// TwinCAT 3 PLC project PLC
// ProgramVersion: 3.1.4023.0
// libraries:
//   Tc2_Standard, * (Beckhoff Automation GmbH)
//   Tc2_System, * (Beckhoff Automation GmbH)
//   Tc3_Module, * (Beckhoff Automation GmbH)
// project tree:
//   / PlcTask.TcTTO
//   POUs/ MAIN.TcPOU
//   DUTs/IO/PdoEntries/ Status_9847B4EF.TcDUT, Status_BA3D1C5D.TcDUT, Status_F2CE6D91.TcDUT, Control_EBEDCF76.TcDUT, FSOE_BBDEEE9E.TcDUT, FSOE_BAC7BF21.TcDUT, FSOE_39DE0EE0.TcDUT, FSOE_3E4279E1.TcDUT, FSOE_BAA7477B.TcDUT, FSOE_CEFF8C56.TcDUT, FSOE_E251F244.TcDUT, FSOE_CDFABDDF.TcDUT
//   DUTs/IO/PDOs/ InfoData_6F19DB2B.TcDUT, ID_07C9D28F.TcDUT, WcState_9091E0EB.TcDUT, Status_Us_B1E819A2.TcDUT, Status_Up_B1E819A2.TcDUT, Channel_830843C1.TcDUT, Channel_42CA91F7.TcDUT, WcState_0B2B16F9.TcDUT, MMS_Device_Inputs_ADC3123E.TcDUT, MMS_Acceleration_Status_11769099.TcDUT, MMS_Acceleration_X_Axis_80E77D6A.TcDUT, MMS_Acceleration_Y_Axis_80E77D6A.TcDUT, MMS_Acceleration_Z_Axis_80E77D6A.TcDUT, MMS_Acceleration_Timestamp_8B9FE1A2.TcDUT, MMS_Voltage_Us_In_Inputs_60D55C72.TcDUT, MMS_Voltage_Up_In_Inputs_60D55C72.TcDUT, MMS_Voltage_Up_Out_Inputs_60D55C72.TcDUT, MMS_Device_Outputs_E6E6F9D1.TcDUT, InfoData_BEF6B88E.TcDUT, FSoE_Inputs_9283FC69.TcDUT, FSoE_Outputs_79E75DAB.TcDUT, Outputs_63C46CC8.TcDUT, FSLOGIC_Inputs_EEE9388E.TcDUT, EMPTY_STRUCTURE.TcDUT, WcState_B516A264.TcDUT, InfoData_32EB74EA.TcDUT, Module_1_FSoE_BE928FF7.TcDUT, Module_2_FSOUT_E84B1B00.TcDUT, Module_3_FSLOGIC_DEAB4522.TcDUT, FSoE_Inputs_6CB74C4A.TcDUT, FSoE_Outputs_D8082339.TcDUT, Outputs_D994E0F9.TcDUT, Module_1_FSoE_042BAFD3.TcDUT, Module_2_FSOUT_8B7AA8A2.TcDUT, FSoE_Inputs_905C1934.TcDUT, FSoE_Outputs_77F9785A.TcDUT, Module_1_FSoE_7E6C60DE.TcDUT, FSoE_Inputs_A1F422BE.TcDUT, FSoE_Outputs_37DEC564.TcDUT, Module_1_FSoE_B78AD590.TcDUT, InfoData_E68C61CD.TcDUT, InfoData_2A97D6CF.TcDUT, Inputs_25A0042B.TcDUT, Outputs_2397A10E.TcDUT
//   DUTs/IO/Boxes/ EK1100_1FC0878B.TcDUT, EK1122_1FC0878B.TcDUT, EK1101_957D888F.TcDUT, EK1110_1FC0878B.TcDUT, EK1121_1FC0878B.TcDUT, EK1200_013D0B49.TcDUT, EK1300_6BC01D14.TcDUT, EK1322_6BC01D14.TcDUT, EK1310_6BC01D14.TcDUT, EK1501_957D888F.TcDUT, EK1541_957D888F.TcDUT, EK1561_1FC0878B.TcDUT, EK1521_1FC0878B.TcDUT, EK1814_F6D9A8D1.TcDUT, EK1818_6B19C24E.TcDUT, EK1828_56D6F887.TcDUT, EK1828_E2806B95.TcDUT, EKM1101_7F417622.TcDUT, EK1960_14394C51.TcDUT, EK1960_9900B192.TcDUT, EK1960_BAE25DEC.TcDUT, EK1960_2415CDAE.TcDUT
//   DUTs/IO/Devices/ SyncUnitTask_2D604ED5.TcDUT, SyncUnitTasks_6FEB8257.TcDUT, SyncUnits_99E584AF.TcDUT
//   DUTs/IO/Topology/ Beckhoff_EK11xxEK1122_42F1D1D1.TcDUT, Beckhoff_EK11xx_811529C6.TcDUT, Beckhoff_EK12xxEK1122_F8B8118B.TcDUT, Beckhoff_EK12xx_F07DE953.TcDUT, Beckhoff_EK13xxEK1122_30D1B042.TcDUT, Beckhoff_EK13xx_7663BCA8.TcDUT, Beckhoff_EK15xxEK1122_1A424B62.TcDUT, Beckhoff_EK15xx_47CB6E2F.TcDUT, Beckhoff_EK18xxEK1122_F7FACD4D.TcDUT, Beckhoff_EK18xx_88ED272B.TcDUT, Beckhoff_EKM1xxxEK1122_F03648A5.TcDUT, Beckhoff_EKM1xxx_245084ED.TcDUT, Beckhoff_EKx9xxEK1122_41BF98AA.TcDUT, Beckhoff_EKx9xx_36A98EAE.TcDUT, Beckhoff_EKxxxx_0080EK1122_9CBA35F2.TcDUT, Beckhoff_EKxxxx_0080_9DDEF925.TcDUT, EtherCAT_Master_EKxxxx_2095F716.TcDUT
//   DUTs/IO/Base/ EtcSlaveBase_82538BE2.TcDUT, EtcSlaveBase_82538BE2.TcDUT, EtcSlaveBase_82538BE2.TcDUT, EtcSlaveTerminalBase_947E5A46.TcDUT, EtcSlaveBoxBase_77A0E4A7.TcDUT, EtcSlaveEndTerminalBase_866C7F0C.TcDUT, InputBase_8311D824.TcDUT, OutputBase_10CEE7DE.TcDUT, EtcMasterBase_62654B43.TcDUT
//   GVLs/ GVL_iXlinker.TcGVL
// real-time tasks:
//   TASK PlcTask: cycle T#10ms, priority 20, ADS port 350
// I/O:
//   DEVICE EtherCAT_Master_EKxxxx, AmsNetId 172.20.30.238.8.1
//     Beckhoff EK11xx [EK1100 EtherCAT Coupler (2A E-Bus)]
//       Beckhoff EK11xxEK1122 [EK1122 2 port EtherCAT junction]
//         Beckhoff EK11xxsub EK1100 [EK1100 EtherCAT Coupler (2A E-Bus)]
//         A_0001(EK1100-0000-0000) [EK1100 EtherCAT Coupler (0.5A E-Bus)]
//         A_0002(EK1100-0000-0001) [EK1100 EtherCAT Coupler (2A E-Bus)]
//         A_0003(EK1100-0000-0016) [EK1100 EtherCAT Coupler (2A E-Bus)]
//         A_0004(EK1100-0000-0017) [EK1100 EtherCAT Coupler (2A E-Bus)]
//         A_0005(EK1100-0000-0018) [EK1100 EtherCAT Coupler (2A E-Bus)]
//         A_0006(EK1100-0008-0016) [EK1100-0008 EtherCAT Coupler M8 (2A E-Bus)]
//         A_0009(EK1101-0000-0016) [EK1101 EtherCAT Coupler (2A E-Bus, ID switch)]
//         A_0010(EK1101-0000-0017) [EK1101 EtherCAT Coupler (2A E-Bus, ID switch)]
//         A_0011(EK1101-0000-0018) [EK1101 EtherCAT Coupler (2A E-Bus, ID switch)]
//         A_0012(EK1101-0008-0016) [EK1101-0008 EtherCAT Coupler M8 (2A E-Bus, ID switch)]
//         A_0013(EK1101-0010-0016) [EK1101-0010 EtherCAT Coupler (2A E-Bus, ID switch, Extended Distance)]
//         A_0008(EK1100-0030-0017) [EK1100-0030 EtherCAT Coupler (2A E-Bus, 4kV galv. iso.)]
//         A_0007(EK1100-0030-0016) [EK1100-0030 EtherCAT Coupler (2A E-Bus, 4kV galv. iso.)]
//       A_0018(EK1110-0043-0016) [EK1110-0043 EtherCAT EJ coupler]
//       A_0024(EK1122-0008-0016) [EK1122-0008 2 port EtherCAT junction M8]
//       A_0023(EK1122-0000-0018) [EK1122 2 port EtherCAT junction]
//       A_0022(EK1122-0000-0017) [EK1122 2 port EtherCAT junction]
//       A_0021(EK1122-0000-0016) [EK1122 2 port EtherCAT junction]
//       A_0020(EK1121-0010-0016) [EK1121-0010 1 port EtherCAT junction (Extended Distance)]
//       A_0019(EK1110-0044-0016) [EK1110-0044 EtherCAT EJ coupler]
//       A_0017(EK1110-0008-0016) [EK1110-0008 EtherCAT extension M8]
//       A_0016(EK1110-0000-0017) [EK1110 EtherCAT extension]
//       A_0015(EK1110-0000-0016) [EK1110 EtherCAT extension]
//       A_0014(EK1110-0000-0000) [EK1110 EtherCAT extension]
//     Beckhoff EK12xx [EK1100 EtherCAT Coupler (2A E-Bus)]
//       Beckhoff EK12xxEK1122 [EK1122 2 port EtherCAT junction]
//         Beckhoff EK12xxsub EK1100 [EK1100 EtherCAT Coupler (2A E-Bus)]
//         A_0002(EK1200-7000-0000) [EK1200-7000 EtherCAT Power supply (1,5A E-Bus)]
//         A_0001(EK1200-5000-0000) [EK1200-5000 EtherCAT Power supply (2A E-Bus)]
//     Beckhoff EK13xx [EK1100 EtherCAT Coupler (2A E-Bus)]
//       Beckhoff EK13xxEK1122 [EK1122 2 port EtherCAT junction]
//         Beckhoff EK13xxsub EK1100 [EK1100 EtherCAT Coupler (2A E-Bus)]
//         A_0001(EK1300-0000-0017) [EK1300 EtherCAT P Coupler (2A E-Bus)]
//       A_0003(EK1322-0000-0017) [EK1322 2-port EtherCAT P junction with feed-in]
//       A_0002(EK1310-0000-0017) [EK1310 EtherCAT P extension with feed-in]
//     Beckhoff EK15xx [EK1100 EtherCAT Coupler (2A E-Bus)]
//       Beckhoff EK15xxEK1122 [EK1122 2 port EtherCAT junction]
//         Beckhoff EK15xxsub EK1100 [EK1100 EtherCAT Coupler (2A E-Bus)]
//         A_0001(EK1501-0000-0016) [EK1501 EtherCAT Coupler (2A E-Bus, FX-MultiMode, ID switch)]
//         A_0002(EK1501-0000-0017) [EK1501 EtherCAT Coupler (2A E-Bus, FX-MultiMode, ID switch)]
//         A_0003(EK1501-0000-0018) [EK1501 EtherCAT Coupler (2A E-Bus, FX-MultiMode, ID switch)]
//         A_0004(EK1501-0000-0019) [EK1501 EtherCAT Coupler (2A E-Bus, FX-MultiMode, ID switch)]
//         A_0005(EK1501-0010-0016) [EK1501-0010 EtherCAT Coupler (2A E-Bus, FX-SingleMode, ID switch)]
//         A_0006(EK1501-0010-0017) [EK1501-0010 EtherCAT Coupler (2A E-Bus, FX-SingleMode, ID switch)]
//         A_0007(EK1501-0010-0018) [EK1501-0010 EtherCAT Coupler (2A E-Bus, FX-SingleMode, ID switch)]
//         A_0008(EK1501-0100-0016) [EK1501-0100 EtherCAT Coupler (2A E-Bus, FX-MultiMode, media converter, ID switch)]
//         A_0020(EK1541-0000-0016) [EK1541 EtherCAT Coupler (2A E-Bus, POF, ID switch)]
//         A_0021(EK1541-0000-0017) [EK1541 EtherCAT Coupler (2A E-Bus, POF, ID switch)]
//         A_0022(EK1541-0000-0018) [EK1541 EtherCAT Coupler (2A E-Bus, POF, ID switch)]
//       A_0025(EK1561-0000-0018) [EK1561 1 port EtherCAT junction (POF)]
//       A_0024(EK1561-0000-0017) [EK1561 1 port EtherCAT junction (POF)]
//       A_0023(EK1561-0000-0016) [EK1561 1 port EtherCAT junction (POF)]
//       A_0019(EK1521-0010-0020) [EK1521-0010 1 port EtherCAT junction (FX-SingleMode)]
//       A_0018(EK1521-0010-0019) [EK1521-0010 1 port EtherCAT junction (FX-SingleMode)]
//       A_0017(EK1521-0010-0018) [EK1521-0010 1 port EtherCAT junction (FX-SingleMode)]
//       A_0016(EK1521-0010-0017) [EK1521-0010 1 port EtherCAT junction (FX-SingleMode)]
//       A_0015(EK1521-0010-0016) [EK1521-0010 1 port EtherCAT junction (FX-SingleMode)]
//       A_0014(EK1521-0000-0021) [EK1521 1 port EtherCAT junction (FX-MultiMode)]
//       A_0013(EK1521-0000-0020) [EK1521 1 port EtherCAT junction (FX-MultiMode)]
//       A_0012(EK1521-0000-0019) [EK1521 1 port EtherCAT junction (FX-MultiMode)]
//       A_0011(EK1521-0000-0018) [EK1521 1 port EtherCAT junction (FX-MultiMode)]
//       A_0010(EK1521-0000-0017) [EK1521 1 port EtherCAT junction (FX-MultiMode)]
//       A_0009(EK1521-0000-0016) [EK1521 1 port EtherCAT junction (FX-MultiMode)]
//     Beckhoff EK18xx [EK1100 EtherCAT Coupler (2A E-Bus)]
//       Beckhoff EK18xxEK1122 [EK1122 2 port EtherCAT junction]
//         Beckhoff EK18xxsub EK1100 [EK1100 EtherCAT Coupler (2A E-Bus)]
//         A_0001(EK1814-0000-0016) [EK1814 EtherCAT IO-Coupler  (0,5A E-Bus, 4 Ch. Dig. In, 3ms, 4 Ch. Dig. Out 24V, 0,5A)]
//         A_0002(EK1814-0000-0017) [EK1814 EtherCAT IO-Coupler  (1A E-Bus, 4 Ch. Dig. In, 3ms, 4 Ch. Dig. Out 24V, 0,5A)]
//         A_0003(EK1814-0000-0018) [EK1814 EtherCAT IO-Coupler  (1A E-Bus, 4 Ch. Dig. In, 3ms, 4 Ch. Dig. Out 24V, 0,5A)]
//         A_0004(EK1814-0000-0019) [EK1814 EtherCAT IO-Coupler  (1A E-Bus, 4 Ch. Dig. In, 3ms, 4 Ch. Dig. Out 24V, 0,5A)]
//         A_0005(EK1818-0000-0016) [EK1818 EtherCAT IO-Coupler  (1A E-Bus, 8 Ch. Dig. In, 3ms, 4 Ch. Dig. Out 24V, 0,5A)]
//         A_0006(EK1818-0000-0017) [EK1818 EtherCAT IO-Coupler  (1A E-Bus, 8 Ch. Dig. In, 3ms, 4 Ch. Dig. Out 24V, 0,5A)]
//         A_0007(EK1818-0000-0018) [EK1818 EtherCAT IO-Coupler  (1A E-Bus, 8 Ch. Dig. In, 3ms, 4 Ch. Dig. Out 24V, 0,5A)]
//         A_0008(EK1828-0000-0016) [EK1828 EtherCAT IO-Coupler  (1A E-Bus, 4 Ch. Dig. In, 3ms, 8 Ch. Dig. Out 24V, 0,5A)]
//         A_0009(EK1828-0000-0017) [EK1828 EtherCAT IO-Coupler  (1A E-Bus, 4 Ch. Dig. In, 3ms, 8 Ch. Dig. Out 24V, 0,5A)]
//         A_0010(EK1828-0000-0018) [EK1828 EtherCAT IO-Coupler  (1A E-Bus, 4 Ch. Dig. In, 3ms, 8 Ch. Dig. Out 24V, 0,5A)]
//         A_0011(EK1828-0010-0016) [EK1828-0010 EtherCAT IO-Coupler  (1A E-Bus, 8 Ch. Dig. Out 24V, 0,5A)]
//         A_0012(EK1828-0010-0017) [EK1828-0010 EtherCAT IO-Coupler  (1A E-Bus, 8 Ch. Dig. Out 24V, 0,5A)]
//         A_0013(EK1828-0010-0018) [EK1828-0010 EtherCAT IO-Coupler  (1A E-Bus, 8 Ch. Dig. Out 24V, 0,5A)]
//     Beckhoff EKM1xxx [EK1100 EtherCAT Coupler (2A E-Bus)]
//       Beckhoff EKM1xxxEK1122 [EK1122 2 port EtherCAT junction]
//         Beckhoff EKM1xxxsub EK1100 [EK1100 EtherCAT Coupler (2A E-Bus)]
//         A_0001(EKM1101-0000-0016) [EKM1101 EtherCAT Coupler  (2A E-Bus, ID switch, Diagnostics, isolated)]
//         A_0002(EKM1101-0000-0017) [EKM1101 EtherCAT Coupler  (2A E-Bus, ID switch, Diagnostics, isolated)]
//         A_0003(EKM1101-0000-0018) [EKM1101 EtherCAT Coupler  (2A E-Bus, ID switch, Diagnostics, isolated)]
//         A_0004(EKM1101-0000-0019) [EKM1101 EtherCAT Coupler  (2A E-Bus, ID switch, Diagnostics, isolated)]
//         A_0005(EKM1101-0000-0020) [EKM1101 EtherCAT Coupler  (2A E-Bus, ID switch, Diagnostics, isolated)]
//     Beckhoff EKx9xx [EK1100 EtherCAT Coupler (2A E-Bus)]
//       Beckhoff EKx9xxEK1122 [EK1122 2 port EtherCAT junction]
//         Beckhoff EKx9xxsub EK1100 [EK1100 EtherCAT Coupler (2A E-Bus)]
//         A_0001(EK1960-0000-0019) [EK1960-0000 TwinSAFE-Compact-Controller (RJ45)]
//           modules: Module 1 (FSoE), Module 2 (FSOUT), Module 3 (FSLOGIC)
//         A_0002(EK1960-0000-0021) [EK1960-0000 TwinSAFE-Compact-Controller (RJ45)]
//           modules: Module 1 (FSoE), Module 2 (FSOUT), Module 3 (FSLOGIC)
//         A_0003(EK1960-0008-0019) [EK1960-0008 TwinSAFE-Compact-Controller (M8)]
//           modules: Module 1 (FSoE), Module 2 (FSOUT), Module 3 (FSLOGIC)
//         A_0004(EK1960-0008-0021) [EK1960-0008 TwinSAFE-Compact-Controller (M8)]
//           modules: Module 1 (FSoE), Module 2 (FSOUT), Module 3 (FSLOGIC)
//         A_0005(EK1960-2600-0019) [EK1960-2600 TwinSAFE-Compact-Controller (4 x Relay, RJ45)]
//           modules: Module 1 (FSoE), Module 2 (FSOUT), Module 3 (FSLOGIC)
//         A_0006(EK1960-2600-0021) [EK1960-2600 TwinSAFE-Compact-Controller (4 x Relay, RJ45)]
//           modules: Module 1 (FSoE), Module 2 (FSOUT), Module 3 (FSLOGIC)
//         A_0007(EK1960-2608-0019) [EK1960-2608 TwinSAFE-Compact-Controller (4 x Relay, M8)]
//           modules: Module 1 (FSoE), Module 2 (FSOUT), Module 3 (FSLOGIC)
//         A_0008(EK1960-2608-0021) [EK1960-2608 TwinSAFE-Compact-Controller (4 x Relay, M8)]
//           modules: Module 1 (FSoE), Module 2 (FSOUT), Module 3 (FSLOGIC)
//     Beckhoff EKxxxx-0080 [EK1100 EtherCAT Coupler (2A E-Bus)]
//       Beckhoff EKxxxx-0080EK1122 [EK1122 2 port EtherCAT junction]
//         Beckhoff EKxxxx-0080sub EK1100 [EK1100 EtherCAT Coupler (2A E-Bus)]
//       A_0006(EK1122-0080-0019) [EK1122-0080 2 port EtherCAT junction (Fast Hot Connect)]
//       A_0005(EK1122-0080-0018) [EK1122-0080 2 port EtherCAT junction (Fast Hot Connect)]
//       A_0004(EK1122-0080-0017) [EK1122-0080 2 port EtherCAT junction (Fast Hot Connect)]
// variable links:
//   PLC/PLC Instance <-> EtherCAT Master EKxxxx/Beckhoff EK11xx
//     PlcTask Inputs/GVL_iXlinker.EtherCAT_Master_EKxxxx.Beckhoff_EK11xx.InfoData.State <-> InfoData/State
//   PLC/PLC Instance <-> EtherCAT Master EKxxxx/Beckhoff EK11xx/Beckhoff EK11xxEK1122
//     PlcTask Inputs/GVL_iXlinker.EtherCAT_Master_EKxxxx.Beckhoff_EK11xx.Beckhoff_EK11xxEK1122.InfoData.State <-> InfoData/State
//   PLC/PLC Instance <-> EtherCAT Master EKxxxx/Beckhoff EK11xx/Beckhoff EK11xxEK1122/Beckhoff EK11xxsub EK1100
//     PlcTask Inputs/GVL_iXlinker.EtherCAT_Master_EKxxxx.Beckhoff_EK11xx.Beckhoff_EK11xxEK1122.Beckhoff_EK11xxsub_EK1100.InfoData.State <-> InfoData/State
//   PLC/PLC Instance <-> EtherCAT Master EKxxxx/Beckhoff EK11xx/Beckhoff EK11xxEK1122/A_0001(EK1100-0000-0000)
//     PlcTask Inputs/GVL_iXlinker.EtherCAT_Master_EKxxxx.Beckhoff_EK11xx.Beckhoff_EK11xxEK1122.A_0001_EK1100_0000_0000.InfoData.State <-> InfoData/State
//   PLC/PLC Instance <-> EtherCAT Master EKxxxx/Beckhoff EK11xx/Beckhoff EK11xxEK1122/A_0002(EK1100-0000-0001)
//     PlcTask Inputs/GVL_iXlinker.EtherCAT_Master_EKxxxx.Beckhoff_EK11xx.Beckhoff_EK11xxEK1122.A_0002_EK1100_0000_0001.InfoData.State <-> InfoData/State
//   PLC/PLC Instance <-> EtherCAT Master EKxxxx/Beckhoff EK11xx/Beckhoff EK11xxEK1122/A_0003(EK1100-0000-0016)
//     PlcTask Inputs/GVL_iXlinker.EtherCAT_Master_EKxxxx.Beckhoff_EK11xx.Beckhoff_EK11xxEK1122.A_0003_EK1100_0000_0016.InfoData.State <-> InfoData/State
//   PLC/PLC Instance <-> EtherCAT Master EKxxxx/Beckhoff EK11xx/Beckhoff EK11xxEK1122/A_0004(EK1100-0000-0017)
//     PlcTask Inputs/GVL_iXlinker.EtherCAT_Master_EKxxxx.Beckhoff_EK11xx.Beckhoff_EK11xxEK1122.A_0004_EK1100_0000_0017.InfoData.State <-> InfoData/State
//   PLC/PLC Instance <-> EtherCAT Master EKxxxx/Beckhoff EK11xx/Beckhoff EK11xxEK1122/A_0005(EK1100-0000-0018)
//     PlcTask Inputs/GVL_iXlinker.EtherCAT_Master_EKxxxx.Beckhoff_EK11xx.Beckhoff_EK11xxEK1122.A_0005_EK1100_0000_0018.InfoData.State <-> InfoData/State
//   PLC/PLC Instance <-> EtherCAT Master EKxxxx/Beckhoff EK11xx/Beckhoff EK11xxEK1122/A_0006(EK1100-0008-0016)
//     PlcTask Inputs/GVL_iXlinker.EtherCAT_Master_EKxxxx.Beckhoff_EK11xx.Beckhoff_EK11xxEK1122.A_0006_EK1100_0008_0016.InfoData.State <-> InfoData/State
//   PLC/PLC Instance <-> EtherCAT Master EKxxxx/Beckhoff EK11xx/Beckhoff EK11xxEK1122/A_0009(EK1101-0000-0016)
//     PlcTask Inputs/GVL_iXlinker.EtherCAT_Master_EKxxxx.Beckhoff_EK11xx.Beckhoff_EK11xxEK1122.A_0009_EK1101_0000_0016.ID.ID <-> ID/ID
//     PlcTask Inputs/GVL_iXlinker.EtherCAT_Master_EKxxxx.Beckhoff_EK11xx.Beckhoff_EK11xxEK1122.A_0009_EK1101_0000_0016.WcState.WcState <-> WcState/WcState
//     PlcTask Inputs/GVL_iXlinker.EtherCAT_Master_EKxxxx.Beckhoff_EK11xx.Beckhoff_EK11xxEK1122.A_0009_EK1101_0000_0016.WcState.InputToggle <-> WcState/InputToggle
//     PlcTask Inputs/GVL_iXlinker.EtherCAT_Master_EKxxxx.Beckhoff_EK11xx.Beckhoff_EK11xxEK1122.A_0009_EK1101_0000_0016.InfoData.State <-> InfoData/State
//   PLC/PLC Instance <-> EtherCAT Master EKxxxx/Beckhoff EK11xx/Beckhoff EK11xxEK1122/A_0010(EK1101-0000-0017)
//     PlcTask Inputs/GVL_iXlinker.EtherCAT_Master_EKxxxx.Beckhoff_EK11xx.Beckhoff_EK11xxEK1122.A_0010_EK1101_0000_0017.ID.ID <-> ID/ID
//     PlcTask Inputs/GVL_iXlinker.EtherCAT_Master_EKxxxx.Beckhoff_EK11xx.Beckhoff_EK11xxEK1122.A_0010_EK1101_0000_0017.WcState.WcState <-> WcState/WcState
//     PlcTask Inputs/GVL_iXlinker.EtherCAT_Master_EKxxxx.Beckhoff_EK11xx.Beckhoff_EK11xxEK1122.A_0010_EK1101_0000_0017.WcState.InputToggle <-> WcState/InputToggle
//     PlcTask Inputs/GVL_iXlinker.EtherCAT_Master_EKxxxx.Beckhoff_EK11xx.Beckhoff_EK11xxEK1122.A_0010_EK1101_0000_0017.InfoData.State <-> InfoData/State
//   PLC/PLC Instance <-> EtherCAT Master EKxxxx/Beckhoff EK11xx/Beckhoff EK11xxEK1122/A_0011(EK1101-0000-0018)
//     PlcTask Inputs/GVL_iXlinker.EtherCAT_Master_EKxxxx.Beckhoff_EK11xx.Beckhoff_EK11xxEK1122.A_0011_EK1101_0000_0018.ID.ID <-> ID/ID
//     PlcTask Inputs/GVL_iXlinker.EtherCAT_Master_EKxxxx.Beckhoff_EK11xx.Beckhoff_EK11xxEK1122.A_0011_EK1101_0000_0018.WcState.WcState <-> WcState/WcState
//     PlcTask Inputs/GVL_iXlinker.EtherCAT_Master_EKxxxx.Beckhoff_EK11xx.Beckhoff_EK11xxEK1122.A_0011_EK1101_0000_0018.WcState.InputToggle <-> WcState/InputToggle
//     PlcTask Inputs/GVL_iXlinker.EtherCAT_Master_EKxxxx.Beckhoff_EK11xx.Beckhoff_EK11xxEK1122.A_0011_EK1101_0000_0018.InfoData.State <-> InfoData/State
//   PLC/PLC Instance <-> EtherCAT Master EKxxxx/Beckhoff EK11xx/Beckhoff EK11xxEK1122/A_0012(EK1101-0008-0016)
//     PlcTask Inputs/GVL_iXlinker.EtherCAT_Master_EKxxxx.Beckhoff_EK11xx.Beckhoff_EK11xxEK1122.A_0012_EK1101_0008_0016.ID.ID <-> ID/ID
//     PlcTask Inputs/GVL_iXlinker.EtherCAT_Master_EKxxxx.Beckhoff_EK11xx.Beckhoff_EK11xxEK1122.A_0012_EK1101_0008_0016.WcState.WcState <-> WcState/WcState
//     PlcTask Inputs/GVL_iXlinker.EtherCAT_Master_EKxxxx.Beckhoff_EK11xx.Beckhoff_EK11xxEK1122.A_0012_EK1101_0008_0016.WcState.InputToggle <-> WcState/InputToggle
//     PlcTask Inputs/GVL_iXlinker.EtherCAT_Master_EKxxxx.Beckhoff_EK11xx.Beckhoff_EK11xxEK1122.A_0012_EK1101_0008_0016.InfoData.State <-> InfoData/State
//   PLC/PLC Instance <-> EtherCAT Master EKxxxx/Beckhoff EK11xx/Beckhoff EK11xxEK1122/A_0013(EK1101-0010-0016)
//     PlcTask Inputs/GVL_iXlinker.EtherCAT_Master_EKxxxx.Beckhoff_EK11xx.Beckhoff_EK11xxEK1122.A_0013_EK1101_0010_0016.ID.ID <-> ID/ID
//     PlcTask Inputs/GVL_iXlinker.EtherCAT_Master_EKxxxx.Beckhoff_EK11xx.Beckhoff_EK11xxEK1122.A_0013_EK1101_0010_0016.WcState.WcState <-> WcState/WcState
//     PlcTask Inputs/GVL_iXlinker.EtherCAT_Master_EKxxxx.Beckhoff_EK11xx.Beckhoff_EK11xxEK1122.A_0013_EK1101_0010_0016.WcState.InputToggle <-> WcState/InputToggle
//     PlcTask Inputs/GVL_iXlinker.EtherCAT_Master_EKxxxx.Beckhoff_EK11xx.Beckhoff_EK11xxEK1122.A_0013_EK1101_0010_0016.InfoData.State <-> InfoData/State
//   PLC/PLC Instance <-> EtherCAT Master EKxxxx/Beckhoff EK11xx/Beckhoff EK11xxEK1122/A_0008(EK1100-0030-0017)
//     PlcTask Inputs/GVL_iXlinker.EtherCAT_Master_EKxxxx.Beckhoff_EK11xx.Beckhoff_EK11xxEK1122.A_0008_EK1100_0030_0017.InfoData.State <-> InfoData/State
//   PLC/PLC Instance <-> EtherCAT Master EKxxxx/Beckhoff EK11xx/Beckhoff EK11xxEK1122/A_0007(EK1100-0030-0016)
//     PlcTask Inputs/GVL_iXlinker.EtherCAT_Master_EKxxxx.Beckhoff_EK11xx.Beckhoff_EK11xxEK1122.A_0007_EK1100_0030_0016.InfoData.State <-> InfoData/State
//   PLC/PLC Instance <-> EtherCAT Master EKxxxx/Beckhoff EK11xx/A_0018(EK1110-0043-0016)
//     PlcTask Inputs/GVL_iXlinker.EtherCAT_Master_EKxxxx.Beckhoff_EK11xx.A_0018_EK1110_0043_0016.InfoData.State <-> InfoData/State
//   PLC/PLC Instance <-> EtherCAT Master EKxxxx/Beckhoff EK11xx/A_0024(EK1122-0008-0016)
//     PlcTask Inputs/GVL_iXlinker.EtherCAT_Master_EKxxxx.Beckhoff_EK11xx.A_0024_EK1122_0008_0016.InfoData.State <-> InfoData/State
//   PLC/PLC Instance <-> EtherCAT Master EKxxxx/Beckhoff EK11xx/A_0023(EK1122-0000-0018)
//     PlcTask Inputs/GVL_iXlinker.EtherCAT_Master_EKxxxx.Beckhoff_EK11xx.A_0023_EK1122_0000_0018.InfoData.State <-> InfoData/State
//   PLC/PLC Instance <-> EtherCAT Master EKxxxx/Beckhoff EK11xx/A_0022(EK1122-0000-0017)
//     PlcTask Inputs/GVL_iXlinker.EtherCAT_Master_EKxxxx.Beckhoff_EK11xx.A_0022_EK1122_0000_0017.InfoData.State <-> InfoData/State
//   PLC/PLC Instance <-> EtherCAT Master EKxxxx/Beckhoff EK11xx/A_0021(EK1122-0000-0016)
//     PlcTask Inputs/GVL_iXlinker.EtherCAT_Master_EKxxxx.Beckhoff_EK11xx.A_0021_EK1122_0000_0016.InfoData.State <-> InfoData/State
//   PLC/PLC Instance <-> EtherCAT Master EKxxxx/Beckhoff EK11xx/A_0020(EK1121-0010-0016)
//     PlcTask Inputs/GVL_iXlinker.EtherCAT_Master_EKxxxx.Beckhoff_EK11xx.A_0020_EK1121_0010_0016.InfoData.State <-> InfoData/State
//   PLC/PLC Instance <-> EtherCAT Master EKxxxx/Beckhoff EK11xx/A_0019(EK1110-0044-0016)
//     PlcTask Inputs/GVL_iXlinker.EtherCAT_Master_EKxxxx.Beckhoff_EK11xx.A_0019_EK1110_0044_0016.InfoData.State <-> InfoData/State
//   PLC/PLC Instance <-> EtherCAT Master EKxxxx/Beckhoff EK11xx/A_0017(EK1110-0008-0016)
//     PlcTask Inputs/GVL_iXlinker.EtherCAT_Master_EKxxxx.Beckhoff_EK11xx.A_0017_EK1110_0008_0016.InfoData.State <-> InfoData/State
//   PLC/PLC Instance <-> EtherCAT Master EKxxxx/Beckhoff EK11xx/A_0016(EK1110-0000-0017)
//     PlcTask Inputs/GVL_iXlinker.EtherCAT_Master_EKxxxx.Beckhoff_EK11xx.A_0016_EK1110_0000_0017.InfoData.State <-> InfoData/State
//   PLC/PLC Instance <-> EtherCAT Master EKxxxx/Beckhoff EK11xx/A_0015(EK1110-0000-0016)
//     PlcTask Inputs/GVL_iXlinker.EtherCAT_Master_EKxxxx.Beckhoff_EK11xx.A_0015_EK1110_0000_0016.InfoData.State <-> InfoData/State
//   PLC/PLC Instance <-> EtherCAT Master EKxxxx/Beckhoff EK11xx/A_0014(EK1110-0000-0000)
//     PlcTask Inputs/GVL_iXlinker.EtherCAT_Master_EKxxxx.Beckhoff_EK11xx.A_0014_EK1110_0000_0000.InfoData.State <-> InfoData/State
//   PLC/PLC Instance <-> EtherCAT Master EKxxxx/Beckhoff EK12xx
//     PlcTask Inputs/GVL_iXlinker.EtherCAT_Master_EKxxxx.Beckhoff_EK12xx.InfoData.State <-> InfoData/State
//   PLC/PLC Instance <-> EtherCAT Master EKxxxx/Beckhoff EK12xx/Beckhoff EK12xxEK1122
//     PlcTask Inputs/GVL_iXlinker.EtherCAT_Master_EKxxxx.Beckhoff_EK12xx.Beckhoff_EK12xxEK1122.InfoData.State <-> InfoData/State
//   PLC/PLC Instance <-> EtherCAT Master EKxxxx/Beckhoff EK12xx/Beckhoff EK12xxEK1122/Beckhoff EK12xxsub EK1100
//     PlcTask Inputs/GVL_iXlinker.EtherCAT_Master_EKxxxx.Beckhoff_EK12xx.Beckhoff_EK12xxEK1122.Beckhoff_EK12xxsub_EK1100.InfoData.State <-> InfoData/State
//   PLC/PLC Instance <-> EtherCAT Master EKxxxx/Beckhoff EK13xx
//     PlcTask Inputs/GVL_iXlinker.EtherCAT_Master_EKxxxx.Beckhoff_EK13xx.InfoData.State <-> InfoData/State
//   PLC/PLC Instance <-> EtherCAT Master EKxxxx/Beckhoff EK13xx/Beckhoff EK13xxEK1122
//     PlcTask Inputs/GVL_iXlinker.EtherCAT_Master_EKxxxx.Beckhoff_EK13xx.Beckhoff_EK13xxEK1122.InfoData.State <-> InfoData/State
//   PLC/PLC Instance <-> EtherCAT Master EKxxxx/Beckhoff EK13xx/Beckhoff EK13xxEK1122/Beckhoff EK13xxsub EK1100
//     PlcTask Inputs/GVL_iXlinker.EtherCAT_Master_EKxxxx.Beckhoff_EK13xx.Beckhoff_EK13xxEK1122.Beckhoff_EK13xxsub_EK1100.InfoData.State <-> InfoData/State
//   PLC/PLC Instance <-> EtherCAT Master EKxxxx/Beckhoff EK13xx/Beckhoff EK13xxEK1122/A_0001(EK1300-0000-0017)
//     PlcTask Inputs/GVL_iXlinker.EtherCAT_Master_EKxxxx.Beckhoff_EK13xx.Beckhoff_EK13xxEK1122.A_0001_EK1300_0000_0017.Status_Us.Undervoltage <-> Status Us/Undervoltage
//     PlcTask Inputs/GVL_iXlinker.EtherCAT_Master_EKxxxx.Beckhoff_EK13xx.Beckhoff_EK13xxEK1122.A_0001_EK1300_0000_0017.Status_Up.Undervoltage <-> Status Up/Undervoltage
//     PlcTask Inputs/GVL_iXlinker.EtherCAT_Master_EKxxxx.Beckhoff_EK13xx.Beckhoff_EK13xxEK1122.A_0001_EK1300_0000_0017.WcState.WcState <-> WcState/WcState
//     PlcTask Inputs/GVL_iXlinker.EtherCAT_Master_EKxxxx.Beckhoff_EK13xx.Beckhoff_EK13xxEK1122.A_0001_EK1300_0000_0017.WcState.InputToggle <-> WcState/InputToggle
//     PlcTask Inputs/GVL_iXlinker.EtherCAT_Master_EKxxxx.Beckhoff_EK13xx.Beckhoff_EK13xxEK1122.A_0001_EK1300_0000_0017.InfoData.State <-> InfoData/State
//   PLC/PLC Instance <-> EtherCAT Master EKxxxx/Beckhoff EK13xx/A_0003(EK1322-0000-0017)
//     PlcTask Inputs/GVL_iXlinker.EtherCAT_Master_EKxxxx.Beckhoff_EK13xx.A_0003_EK1322_0000_0017.Status_Us.Undervoltage <-> Status Us/Undervoltage
//     PlcTask Inputs/GVL_iXlinker.EtherCAT_Master_EKxxxx.Beckhoff_EK13xx.A_0003_EK1322_0000_0017.Status_Up.Undervoltage <-> Status Up/Undervoltage
//     PlcTask Inputs/GVL_iXlinker.EtherCAT_Master_EKxxxx.Beckhoff_EK13xx.A_0003_EK1322_0000_0017.WcState.WcState <-> WcState/WcState
//     PlcTask Inputs/GVL_iXlinker.EtherCAT_Master_EKxxxx.Beckhoff_EK13xx.A_0003_EK1322_0000_0017.WcState.InputToggle <-> WcState/InputToggle
//     PlcTask Inputs/GVL_iXlinker.EtherCAT_Master_EKxxxx.Beckhoff_EK13xx.A_0003_EK1322_0000_0017.InfoData.State <-> InfoData/State
//   PLC/PLC Instance <-> EtherCAT Master EKxxxx/Beckhoff EK13xx/A_0002(EK1310-0000-0017)
//     PlcTask Inputs/GVL_iXlinker.EtherCAT_Master_EKxxxx.Beckhoff_EK13xx.A_0002_EK1310_0000_0017.Status_Us.Undervoltage <-> Status Us/Undervoltage
//     PlcTask Inputs/GVL_iXlinker.EtherCAT_Master_EKxxxx.Beckhoff_EK13xx.A_0002_EK1310_0000_0017.Status_Up.Undervoltage <-> Status Up/Undervoltage
//     PlcTask Inputs/GVL_iXlinker.EtherCAT_Master_EKxxxx.Beckhoff_EK13xx.A_0002_EK1310_0000_0017.WcState.WcState <-> WcState/WcState
//     PlcTask Inputs/GVL_iXlinker.EtherCAT_Master_EKxxxx.Beckhoff_EK13xx.A_0002_EK1310_0000_0017.WcState.InputToggle <-> WcState/InputToggle
//     PlcTask Inputs/GVL_iXlinker.EtherCAT_Master_EKxxxx.Beckhoff_EK13xx.A_0002_EK1310_0000_0017.InfoData.State <-> InfoData/State
//   PLC/PLC Instance <-> EtherCAT Master EKxxxx/Beckhoff EK15xx
//     PlcTask Inputs/GVL_iXlinker.EtherCAT_Master_EKxxxx.Beckhoff_EK15xx.InfoData.State <-> InfoData/State
//   PLC/PLC Instance <-> EtherCAT Master EKxxxx/Beckhoff EK15xx/Beckhoff EK15xxEK1122
//     PlcTask Inputs/GVL_iXlinker.EtherCAT_Master_EKxxxx.Beckhoff_EK15xx.Beckhoff_EK15xxEK1122.InfoData.State <-> InfoData/State
//   PLC/PLC Instance <-> EtherCAT Master EKxxxx/Beckhoff EK15xx/Beckhoff EK15xxEK1122/Beckhoff EK15xxsub EK1100
//     PlcTask Inputs/GVL_iXlinker.EtherCAT_Master_EKxxxx.Beckhoff_EK15xx.Beckhoff_EK15xxEK1122.Beckhoff_EK15xxsub_EK1100.InfoData.State <-> InfoData/State
//   PLC/PLC Instance <-> EtherCAT Master EKxxxx/Beckhoff EK15xx/Beckhoff EK15xxEK1122/A_0001(EK1501-0000-0016)
//     PlcTask Inputs/GVL_iXlinker.EtherCAT_Master_EKxxxx.Beckhoff_EK15xx.Beckhoff_EK15xxEK1122.A_0001_EK1501_0000_0016.ID.ID <-> ID/ID
//     PlcTask Inputs/GVL_iXlinker.EtherCAT_Master_EKxxxx.Beckhoff_EK15xx.Beckhoff_EK15xxEK1122.A_0001_EK1501_0000_0016.WcState.WcState <-> WcState/WcState
//     PlcTask Inputs/GVL_iXlinker.EtherCAT_Master_EKxxxx.Beckhoff_EK15xx.Beckhoff_EK15xxEK1122.A_0001_EK1501_0000_0016.WcState.InputToggle <-> WcState/InputToggle
//     PlcTask Inputs/GVL_iXlinker.EtherCAT_Master_EKxxxx.Beckhoff_EK15xx.Beckhoff_EK15xxEK1122.A_0001_EK1501_0000_0016.InfoData.State <-> InfoData/State
//   PLC/PLC Instance <-> EtherCAT Master EKxxxx/Beckhoff EK15xx/Beckhoff EK15xxEK1122/A_0002(EK1501-0000-0017)
//     PlcTask Inputs/GVL_iXlinker.EtherCAT_Master_EKxxxx.Beckhoff_EK15xx.Beckhoff_EK15xxEK1122.A_0002_EK1501_0000_0017.ID.ID <-> ID/ID
//     PlcTask Inputs/GVL_iXlinker.EtherCAT_Master_EKxxxx.Beckhoff_EK15xx.Beckhoff_EK15xxEK1122.A_0002_EK1501_0000_0017.WcState.WcState <-> WcState/WcState
//     PlcTask Inputs/GVL_iXlinker.EtherCAT_Master_EKxxxx.Beckhoff_EK15xx.Beckhoff_EK15xxEK1122.A_0002_EK1501_0000_0017.WcState.InputToggle <-> WcState/InputToggle
//     PlcTask Inputs/GVL_iXlinker.EtherCAT_Master_EKxxxx.Beckhoff_EK15xx.Beckhoff_EK15xxEK1122.A_0002_EK1501_0000_0017.InfoData.State <-> InfoData/State
//   PLC/PLC Instance <-> EtherCAT Master EKxxxx/Beckhoff EK15xx/Beckhoff EK15xxEK1122/A_0003(EK1501-0000-0018)
//     PlcTask Inputs/GVL_iXlinker.EtherCAT_Master_EKxxxx.Beckhoff_EK15xx.Beckhoff_EK15xxEK1122.A_0003_EK1501_0000_0018.ID.ID <-> ID/ID
//     PlcTask Inputs/GVL_iXlinker.EtherCAT_Master_EKxxxx.Beckhoff_EK15xx.Beckhoff_EK15xxEK1122.A_0003_EK1501_0000_0018.WcState.WcState <-> WcState/WcState
//     PlcTask Inputs/GVL_iXlinker.EtherCAT_Master_EKxxxx.Beckhoff_EK15xx.Beckhoff_EK15xxEK1122.A_0003_EK1501_0000_0018.WcState.InputToggle <-> WcState/InputToggle
//     PlcTask Inputs/GVL_iXlinker.EtherCAT_Master_EKxxxx.Beckhoff_EK15xx.Beckhoff_EK15xxEK1122.A_0003_EK1501_0000_0018.InfoData.State <-> InfoData/State
//   PLC/PLC Instance <-> EtherCAT Master EKxxxx/Beckhoff EK15xx/Beckhoff EK15xxEK1122/A_0004(EK1501-0000-0019)
//     PlcTask Inputs/GVL_iXlinker.EtherCAT_Master_EKxxxx.Beckhoff_EK15xx.Beckhoff_EK15xxEK1122.A_0004_EK1501_0000_0019.ID.ID <-> ID/ID
//     PlcTask Inputs/GVL_iXlinker.EtherCAT_Master_EKxxxx.Beckhoff_EK15xx.Beckhoff_EK15xxEK1122.A_0004_EK1501_0000_0019.WcState.WcState <-> WcState/WcState
//     PlcTask Inputs/GVL_iXlinker.EtherCAT_Master_EKxxxx.Beckhoff_EK15xx.Beckhoff_EK15xxEK1122.A_0004_EK1501_0000_0019.WcState.InputToggle <-> WcState/InputToggle
//     PlcTask Inputs/GVL_iXlinker.EtherCAT_Master_EKxxxx.Beckhoff_EK15xx.Beckhoff_EK15xxEK1122.A_0004_EK1501_0000_0019.InfoData.State <-> InfoData/State
//   PLC/PLC Instance <-> EtherCAT Master EKxxxx/Beckhoff EK15xx/Beckhoff EK15xxEK1122/A_0005(EK1501-0010-0016)
//     PlcTask Inputs/GVL_iXlinker.EtherCAT_Master_EKxxxx.Beckhoff_EK15xx.Beckhoff_EK15xxEK1122.A_0005_EK1501_0010_0016.ID.ID <-> ID/ID
//     PlcTask Inputs/GVL_iXlinker.EtherCAT_Master_EKxxxx.Beckhoff_EK15xx.Beckhoff_EK15xxEK1122.A_0005_EK1501_0010_0016.WcState.WcState <-> WcState/WcState
//     PlcTask Inputs/GVL_iXlinker.EtherCAT_Master_EKxxxx.Beckhoff_EK15xx.Beckhoff_EK15xxEK1122.A_0005_EK1501_0010_0016.WcState.InputToggle <-> WcState/InputToggle
//     PlcTask Inputs/GVL_iXlinker.EtherCAT_Master_EKxxxx.Beckhoff_EK15xx.Beckhoff_EK15xxEK1122.A_0005_EK1501_0010_0016.InfoData.State <-> InfoData/State
//   PLC/PLC Instance <-> EtherCAT Master EKxxxx/Beckhoff EK15xx/Beckhoff EK15xxEK1122/A_0006(EK1501-0010-0017)
//     PlcTask Inputs/GVL_iXlinker.EtherCAT_Master_EKxxxx.Beckhoff_EK15xx.Beckhoff_EK15xxEK1122.A_0006_EK1501_0010_0017.ID.ID <-> ID/ID
//     PlcTask Inputs/GVL_iXlinker.EtherCAT_Master_EKxxxx.Beckhoff_EK15xx.Beckhoff_EK15xxEK1122.A_0006_EK1501_0010_0017.WcState.WcState <-> WcState/WcState
//     PlcTask Inputs/GVL_iXlinker.EtherCAT_Master_EKxxxx.Beckhoff_EK15xx.Beckhoff_EK15xxEK1122.A_0006_EK1501_0010_0017.WcState.InputToggle <-> WcState/InputToggle
//     PlcTask Inputs/GVL_iXlinker.EtherCAT_Master_EKxxxx.Beckhoff_EK15xx.Beckhoff_EK15xxEK1122.A_0006_EK1501_0010_0017.InfoData.State <-> InfoData/State
//   PLC/PLC Instance <-> EtherCAT Master EKxxxx/Beckhoff EK15xx/Beckhoff EK15xxEK1122/A_0007(EK1501-0010-0018)
//     PlcTask Inputs/GVL_iXlinker.EtherCAT_Master_EKxxxx.Beckhoff_EK15xx.Beckhoff_EK15xxEK1122.A_0007_EK1501_0010_0018.ID.ID <-> ID/ID
//     PlcTask Inputs/GVL_iXlinker.EtherCAT_Master_EKxxxx.Beckhoff_EK15xx.Beckhoff_EK15xxEK1122.A_0007_EK1501_0010_0018.WcState.WcState <-> WcState/WcState
//     PlcTask Inputs/GVL_iXlinker.EtherCAT_Master_EKxxxx.Beckhoff_EK15xx.Beckhoff_EK15xxEK1122.A_0007_EK1501_0010_0018.WcState.InputToggle <-> WcState/InputToggle
//     PlcTask Inputs/GVL_iXlinker.EtherCAT_Master_EKxxxx.Beckhoff_EK15xx.Beckhoff_EK15xxEK1122.A_0007_EK1501_0010_0018.InfoData.State <-> InfoData/State
//   PLC/PLC Instance <-> EtherCAT Master EKxxxx/Beckhoff EK15xx/Beckhoff EK15xxEK1122/A_0008(EK1501-0100-0016)
//     PlcTask Inputs/GVL_iXlinker.EtherCAT_Master_EKxxxx.Beckhoff_EK15xx.Beckhoff_EK15xxEK1122.A_0008_EK1501_0100_0016.ID.ID <-> ID/ID
//     PlcTask Inputs/GVL_iXlinker.EtherCAT_Master_EKxxxx.Beckhoff_EK15xx.Beckhoff_EK15xxEK1122.A_0008_EK1501_0100_0016.WcState.WcState <-> WcState/WcState
//     PlcTask Inputs/GVL_iXlinker.EtherCAT_Master_EKxxxx.Beckhoff_EK15xx.Beckhoff_EK15xxEK1122.A_0008_EK1501_0100_0016.WcState.InputToggle <-> WcState/InputToggle
//     PlcTask Inputs/GVL_iXlinker.EtherCAT_Master_EKxxxx.Beckhoff_EK15xx.Beckhoff_EK15xxEK1122.A_0008_EK1501_0100_0016.InfoData.State <-> InfoData/State
//   PLC/PLC Instance <-> EtherCAT Master EKxxxx/Beckhoff EK15xx/Beckhoff EK15xxEK1122/A_0020(EK1541-0000-0016)
//     PlcTask Inputs/GVL_iXlinker.EtherCAT_Master_EKxxxx.Beckhoff_EK15xx.Beckhoff_EK15xxEK1122.A_0020_EK1541_0000_0016.ID.ID <-> ID/ID
//     PlcTask Inputs/GVL_iXlinker.EtherCAT_Master_EKxxxx.Beckhoff_EK15xx.Beckhoff_EK15xxEK1122.A_0020_EK1541_0000_0016.WcState.WcState <-> WcState/WcState
//     PlcTask Inputs/GVL_iXlinker.EtherCAT_Master_EKxxxx.Beckhoff_EK15xx.Beckhoff_EK15xxEK1122.A_0020_EK1541_0000_0016.WcState.InputToggle <-> WcState/InputToggle
//     PlcTask Inputs/GVL_iXlinker.EtherCAT_Master_EKxxxx.Beckhoff_EK15xx.Beckhoff_EK15xxEK1122.A_0020_EK1541_0000_0016.InfoData.State <-> InfoData/State
//   PLC/PLC Instance <-> EtherCAT Master EKxxxx/Beckhoff EK15xx/Beckhoff EK15xxEK1122/A_0021(EK1541-0000-0017)
//     PlcTask Inputs/GVL_iXlinker.EtherCAT_Master_EKxxxx.Beckhoff_EK15xx.Beckhoff_EK15xxEK1122.A_0021_EK1541_0000_0017.ID.ID <-> ID/ID
//     PlcTask Inputs/GVL_iXlinker.EtherCAT_Master_EKxxxx.Beckhoff_EK15xx.Beckhoff_EK15xxEK1122.A_0021_EK1541_0000_0017.WcState.WcState <-> WcState/WcState
//     PlcTask Inputs/GVL_iXlinker.EtherCAT_Master_EKxxxx.Beckhoff_EK15xx.Beckhoff_EK15xxEK1122.A_0021_EK1541_0000_0017.WcState.InputToggle <-> WcState/InputToggle
//     PlcTask Inputs/GVL_iXlinker.EtherCAT_Master_EKxxxx.Beckhoff_EK15xx.Beckhoff_EK15xxEK1122.A_0021_EK1541_0000_0017.InfoData.State <-> InfoData/State
//   PLC/PLC Instance <-> EtherCAT Master EKxxxx/Beckhoff EK15xx/Beckhoff EK15xxEK1122/A_0022(EK1541-0000-0018)
//     PlcTask Inputs/GVL_iXlinker.EtherCAT_Master_EKxxxx.Beckhoff_EK15xx.Beckhoff_EK15xxEK1122.A_0022_EK1541_0000_0018.ID.ID <-> ID/ID
//     PlcTask Inputs/GVL_iXlinker.EtherCAT_Master_EKxxxx.Beckhoff_EK15xx.Beckhoff_EK15xxEK1122.A_0022_EK1541_0000_0018.WcState.WcState <-> WcState/WcState
//     PlcTask Inputs/GVL_iXlinker.EtherCAT_Master_EKxxxx.Beckhoff_EK15xx.Beckhoff_EK15xxEK1122.A_0022_EK1541_0000_0018.WcState.InputToggle <-> WcState/InputToggle
//     PlcTask Inputs/GVL_iXlinker.EtherCAT_Master_EKxxxx.Beckhoff_EK15xx.Beckhoff_EK15xxEK1122.A_0022_EK1541_0000_0018.InfoData.State <-> InfoData/State
//   PLC/PLC Instance <-> EtherCAT Master EKxxxx/Beckhoff EK15xx/A_0025(EK1561-0000-0018)
//     PlcTask Inputs/GVL_iXlinker.EtherCAT_Master_EKxxxx.Beckhoff_EK15xx.A_0025_EK1561_0000_0018.InfoData.State <-> InfoData/State
//   PLC/PLC Instance <-> EtherCAT Master EKxxxx/Beckhoff EK15xx/A_0024(EK1561-0000-0017)
//     PlcTask Inputs/GVL_iXlinker.EtherCAT_Master_EKxxxx.Beckhoff_EK15xx.A_0024_EK1561_0000_0017.InfoData.State <-> InfoData/State
//   PLC/PLC Instance <-> EtherCAT Master EKxxxx/Beckhoff EK15xx/A_0023(EK1561-0000-0016)
//     PlcTask Inputs/GVL_iXlinker.EtherCAT_Master_EKxxxx.Beckhoff_EK15xx.A_0023_EK1561_0000_0016.InfoData.State <-> InfoData/State
//   PLC/PLC Instance <-> EtherCAT Master EKxxxx/Beckhoff EK15xx/A_0019(EK1521-0010-0020)
//     PlcTask Inputs/GVL_iXlinker.EtherCAT_Master_EKxxxx.Beckhoff_EK15xx.A_0019_EK1521_0010_0020.InfoData.State <-> InfoData/State
//   PLC/PLC Instance <-> EtherCAT Master EKxxxx/Beckhoff EK15xx/A_0018(EK1521-0010-0019)
//     PlcTask Inputs/GVL_iXlinker.EtherCAT_Master_EKxxxx.Beckhoff_EK15xx.A_0018_EK1521_0010_0019.InfoData.State <-> InfoData/State
//   PLC/PLC Instance <-> EtherCAT Master EKxxxx/Beckhoff EK15xx/A_0017(EK1521-0010-0018)
//     PlcTask Inputs/GVL_iXlinker.EtherCAT_Master_EKxxxx.Beckhoff_EK15xx.A_0017_EK1521_0010_0018.InfoData.State <-> InfoData/State
//   PLC/PLC Instance <-> EtherCAT Master EKxxxx/Beckhoff EK15xx/A_0016(EK1521-0010-0017)
//     PlcTask Inputs/GVL_iXlinker.EtherCAT_Master_EKxxxx.Beckhoff_EK15xx.A_0016_EK1521_0010_0017.InfoData.State <-> InfoData/State
//   PLC/PLC Instance <-> EtherCAT Master EKxxxx/Beckhoff EK15xx/A_0015(EK1521-0010-0016)
//     PlcTask Inputs/GVL_iXlinker.EtherCAT_Master_EKxxxx.Beckhoff_EK15xx.A_0015_EK1521_0010_0016.InfoData.State <-> InfoData/State
//   PLC/PLC Instance <-> EtherCAT Master EKxxxx/Beckhoff EK15xx/A_0014(EK1521-0000-0021)
//     PlcTask Inputs/GVL_iXlinker.EtherCAT_Master_EKxxxx.Beckhoff_EK15xx.A_0014_EK1521_0000_0021.InfoData.State <-> InfoData/State
//   PLC/PLC Instance <-> EtherCAT Master EKxxxx/Beckhoff EK15xx/A_0013(EK1521-0000-0020)
//     PlcTask Inputs/GVL_iXlinker.EtherCAT_Master_EKxxxx.Beckhoff_EK15xx.A_0013_EK1521_0000_0020.InfoData.State <-> InfoData/State
//   PLC/PLC Instance <-> EtherCAT Master EKxxxx/Beckhoff EK15xx/A_0012(EK1521-0000-0019)
//     PlcTask Inputs/GVL_iXlinker.EtherCAT_Master_EKxxxx.Beckhoff_EK15xx.A_0012_EK1521_0000_0019.InfoData.State <-> InfoData/State
//   PLC/PLC Instance <-> EtherCAT Master EKxxxx/Beckhoff EK15xx/A_0011(EK1521-0000-0018)
//     PlcTask Inputs/GVL_iXlinker.EtherCAT_Master_EKxxxx.Beckhoff_EK15xx.A_0011_EK1521_0000_0018.InfoData.State <-> InfoData/State
//   PLC/PLC Instance <-> EtherCAT Master EKxxxx/Beckhoff EK15xx/A_0010(EK1521-0000-0017)
//     PlcTask Inputs/GVL_iXlinker.EtherCAT_Master_EKxxxx.Beckhoff_EK15xx.A_0010_EK1521_0000_0017.InfoData.State <-> InfoData/State
//   PLC/PLC Instance <-> EtherCAT Master EKxxxx/Beckhoff EK15xx/A_0009(EK1521-0000-0016)
//     PlcTask Inputs/GVL_iXlinker.EtherCAT_Master_EKxxxx.Beckhoff_EK15xx.A_0009_EK1521_0000_0016.InfoData.State <-> InfoData/State
//   PLC/PLC Instance <-> EtherCAT Master EKxxxx/Beckhoff EK18xx
//     PlcTask Inputs/GVL_iXlinker.EtherCAT_Master_EKxxxx.Beckhoff_EK18xx.InfoData.State <-> InfoData/State
//   PLC/PLC Instance <-> EtherCAT Master EKxxxx/Beckhoff EK18xx/Beckhoff EK18xxEK1122
//     PlcTask Inputs/GVL_iXlinker.EtherCAT_Master_EKxxxx.Beckhoff_EK18xx.Beckhoff_EK18xxEK1122.InfoData.State <-> InfoData/State
//   PLC/PLC Instance <-> EtherCAT Master EKxxxx/Beckhoff EK18xx/Beckhoff EK18xxEK1122/Beckhoff EK18xxsub EK1100
//     PlcTask Inputs/GVL_iXlinker.EtherCAT_Master_EKxxxx.Beckhoff_EK18xx.Beckhoff_EK18xxEK1122.Beckhoff_EK18xxsub_EK1100.InfoData.State <-> InfoData/State
//   PLC/PLC Instance <-> EtherCAT Master EKxxxx/Beckhoff EK18xx/Beckhoff EK18xxEK1122/A_0001(EK1814-0000-0016)
//     PlcTask Inputs/GVL_iXlinker.EtherCAT_Master_EKxxxx.Beckhoff_EK18xx.Beckhoff_EK18xxEK1122.A_0001_EK1814_0000_0016.Channel_1.Input <-> Channel 1/Input
//     PlcTask Inputs/GVL_iXlinker.EtherCAT_Master_EKxxxx.Beckhoff_EK18xx.Beckhoff_EK18xxEK1122.A_0001_EK1814_0000_0016.Channel_2.Input <-> Channel 2/Input
//     PlcTask Inputs/GVL_iXlinker.EtherCAT_Master_EKxxxx.Beckhoff_EK18xx.Beckhoff_EK18xxEK1122.A_0001_EK1814_0000_0016.Channel_3.Input <-> Channel 3/Input
//     PlcTask Inputs/GVL_iXlinker.EtherCAT_Master_EKxxxx.Beckhoff_EK18xx.Beckhoff_EK18xxEK1122.A_0001_EK1814_0000_0016.Channel_4.Input <-> Channel 4/Input
//     PlcTask Outputs/GVL_iXlinker.EtherCAT_Master_EKxxxx.Beckhoff_EK18xx.Beckhoff_EK18xxEK1122.A_0001_EK1814_0000_0016.Channel_5.Output <-> Channel 5/Output
//     PlcTask Outputs/GVL_iXlinker.EtherCAT_Master_EKxxxx.Beckhoff_EK18xx.Beckhoff_EK18xxEK1122.A_0001_EK1814_0000_0016.Channel_6.Output <-> Channel 6/Output
//     PlcTask Outputs/GVL_iXlinker.EtherCAT_Master_EKxxxx.Beckhoff_EK18xx.Beckhoff_EK18xxEK1122.A_0001_EK1814_0000_0016.Channel_7.Output <-> Channel 7/Output
//     PlcTask Outputs/GVL_iXlinker.EtherCAT_Master_EKxxxx.Beckhoff_EK18xx.Beckhoff_EK18xxEK1122.A_0001_EK1814_0000_0016.Channel_8.Output <-> Channel 8/Output
//     PlcTask Inputs/GVL_iXlinker.EtherCAT_Master_EKxxxx.Beckhoff_EK18xx.Beckhoff_EK18xxEK1122.A_0001_EK1814_0000_0016.WcState.WcState <-> WcState/WcState
//     PlcTask Inputs/GVL_iXlinker.EtherCAT_Master_EKxxxx.Beckhoff_EK18xx.Beckhoff_EK18xxEK1122.A_0001_EK1814_0000_0016.WcState.InputToggle <-> WcState/InputToggle
//     PlcTask Inputs/GVL_iXlinker.EtherCAT_Master_EKxxxx.Beckhoff_EK18xx.Beckhoff_EK18xxEK1122.A_0001_EK1814_0000_0016.InfoData.State <-> InfoData/State
//   PLC/PLC Instance <-> EtherCAT Master EKxxxx/Beckhoff EK18xx/Beckhoff EK18xxEK1122/A_0002(EK1814-0000-0017)
//     PlcTask Inputs/GVL_iXlinker.EtherCAT_Master_EKxxxx.Beckhoff_EK18xx.Beckhoff_EK18xxEK1122.A_0002_EK1814_0000_0017.Channel_1.Input <-> Channel 1/Input
//     PlcTask Inputs/GVL_iXlinker.EtherCAT_Master_EKxxxx.Beckhoff_EK18xx.Beckhoff_EK18xxEK1122.A_0002_EK1814_0000_0017.Channel_2.Input <-> Channel 2/Input
//     PlcTask Inputs/GVL_iXlinker.EtherCAT_Master_EKxxxx.Beckhoff_EK18xx.Beckhoff_EK18xxEK1122.A_0002_EK1814_0000_0017.Channel_3.Input <-> Channel 3/Input
//     PlcTask Inputs/GVL_iXlinker.EtherCAT_Master_EKxxxx.Beckhoff_EK18xx.Beckhoff_EK18xxEK1122.A_0002_EK1814_0000_0017.Channel_4.Input <-> Channel 4/Input
//     PlcTask Outputs/GVL_iXlinker.EtherCAT_Master_EKxxxx.Beckhoff_EK18xx.Beckhoff_EK18xxEK1122.A_0002_EK1814_0000_0017.Channel_5.Output <-> Channel 5/Output
//     PlcTask Outputs/GVL_iXlinker.EtherCAT_Master_EKxxxx.Beckhoff_EK18xx.Beckhoff_EK18xxEK1122.A_0002_EK1814_0000_0017.Channel_6.Output <-> Channel 6/Output
//     PlcTask Outputs/GVL_iXlinker.EtherCAT_Master_EKxxxx.Beckhoff_EK18xx.Beckhoff_EK18xxEK1122.A_0002_EK1814_0000_0017.Channel_7.Output <-> Channel 7/Output
//     PlcTask Outputs/GVL_iXlinker.EtherCAT_Master_EKxxxx.Beckhoff_EK18xx.Beckhoff_EK18xxEK1122.A_0002_EK1814_0000_0017.Channel_8.Output <-> Channel 8/Output
//     PlcTask Inputs/GVL_iXlinker.EtherCAT_Master_EKxxxx.Beckhoff_EK18xx.Beckhoff_EK18xxEK1122.A_0002_EK1814_0000_0017.WcState.WcState <-> WcState/WcState
//     PlcTask Inputs/GVL_iXlinker.EtherCAT_Master_EKxxxx.Beckhoff_EK18xx.Beckhoff_EK18xxEK1122.A_0002_EK1814_0000_0017.WcState.InputToggle <-> WcState/InputToggle
//     PlcTask Inputs/GVL_iXlinker.EtherCAT_Master_EKxxxx.Beckhoff_EK18xx.Beckhoff_EK18xxEK1122.A_0002_EK1814_0000_0017.InfoData.State <-> InfoData/State
//   PLC/PLC Instance <-> EtherCAT Master EKxxxx/Beckhoff EK18xx/Beckhoff EK18xxEK1122/A_0003(EK1814-0000-0018)
//     PlcTask Inputs/GVL_iXlinker.EtherCAT_Master_EKxxxx.Beckhoff_EK18xx.Beckhoff_EK18xxEK1122.A_0003_EK1814_0000_0018.Channel_1.Input <-> Channel 1/Input
//     PlcTask Inputs/GVL_iXlinker.EtherCAT_Master_EKxxxx.Beckhoff_EK18xx.Beckhoff_EK18xxEK1122.A_0003_EK1814_0000_0018.Channel_2.Input <-> Channel 2/Input
//     PlcTask Inputs/GVL_iXlinker.EtherCAT_Master_EKxxxx.Beckhoff_EK18xx.Beckhoff_EK18xxEK1122.A_0003_EK1814_0000_0018.Channel_3.Input <-> Channel 3/Input
//     PlcTask Inputs/GVL_iXlinker.EtherCAT_Master_EKxxxx.Beckhoff_EK18xx.Beckhoff_EK18xxEK1122.A_0003_EK1814_0000_0018.Channel_4.Input <-> Channel 4/Input
//     PlcTask Outputs/GVL_iXlinker.EtherCAT_Master_EKxxxx.Beckhoff_EK18xx.Beckhoff_EK18xxEK1122.A_0003_EK1814_0000_0018.Channel_5.Output <-> Channel 5/Output
//     PlcTask Outputs/GVL_iXlinker.EtherCAT_Master_EKxxxx.Beckhoff_EK18xx.Beckhoff_EK18xxEK1122.A_0003_EK1814_0000_0018.Channel_6.Output <-> Channel 6/Output
//     PlcTask Outputs/GVL_iXlinker.EtherCAT_Master_EKxxxx.Beckhoff_EK18xx.Beckhoff_EK18xxEK1122.A_0003_EK1814_0000_0018.Channel_7.Output <-> Channel 7/Output
//     PlcTask Outputs/GVL_iXlinker.EtherCAT_Master_EKxxxx.Beckhoff_EK18xx.Beckhoff_EK18xxEK1122.A_0003_EK1814_0000_0018.Channel_8.Output <-> Channel 8/Output
//     PlcTask Inputs/GVL_iXlinker.EtherCAT_Master_EKxxxx.Beckhoff_EK18xx.Beckhoff_EK18xxEK1122.A_0003_EK1814_0000_0018.WcState.WcState <-> WcState/WcState
//     PlcTask Inputs/GVL_iXlinker.EtherCAT_Master_EKxxxx.Beckhoff_EK18xx.Beckhoff_EK18xxEK1122.A_0003_EK1814_0000_0018.WcState.InputToggle <-> WcState/InputToggle
//     PlcTask Inputs/GVL_iXlinker.EtherCAT_Master_EKxxxx.Beckhoff_EK18xx.Beckhoff_EK18xxEK1122.A_0003_EK1814_0000_0018.InfoData.State <-> InfoData/State
//   PLC/PLC Instance <-> EtherCAT Master EKxxxx/Beckhoff EK18xx/Beckhoff EK18xxEK1122/A_0004(EK1814-0000-0019)
//     PlcTask Inputs/GVL_iXlinker.EtherCAT_Master_EKxxxx.Beckhoff_EK18xx.Beckhoff_EK18xxEK1122.A_0004_EK1814_0000_0019.Channel_1.Input <-> Channel 1/Input
//     PlcTask Inputs/GVL_iXlinker.EtherCAT_Master_EKxxxx.Beckhoff_EK18xx.Beckhoff_EK18xxEK1122.A_0004_EK1814_0000_0019.Channel_2.Input <-> Channel 2/Input
//     PlcTask Inputs/GVL_iXlinker.EtherCAT_Master_EKxxxx.Beckhoff_EK18xx.Beckhoff_EK18xxEK1122.A_0004_EK1814_0000_0019.Channel_3.Input <-> Channel 3/Input
//     PlcTask Inputs/GVL_iXlinker.EtherCAT_Master_EKxxxx.Beckhoff_EK18xx.Beckhoff_EK18xxEK1122.A_0004_EK1814_0000_0019.Channel_4.Input <-> Channel 4/Input
//     PlcTask Outputs/GVL_iXlinker.EtherCAT_Master_EKxxxx.Beckhoff_EK18xx.Beckhoff_EK18xxEK1122.A_0004_EK1814_0000_0019.Channel_5.Output <-> Channel 5/Output
//     PlcTask Outputs/GVL_iXlinker.EtherCAT_Master_EKxxxx.Beckhoff_EK18xx.Beckhoff_EK18xxEK1122.A_0004_EK1814_0000_0019.Channel_6.Output <-> Channel 6/Output
//     PlcTask Outputs/GVL_iXlinker.EtherCAT_Master_EKxxxx.Beckhoff_EK18xx.Beckhoff_EK18xxEK1122.A_0004_EK1814_0000_0019.Channel_7.Output <-> Channel 7/Output
//     PlcTask Outputs/GVL_iXlinker.EtherCAT_Master_EKxxxx.Beckhoff_EK18xx.Beckhoff_EK18xxEK1122.A_0004_EK1814_0000_0019.Channel_8.Output <-> Channel 8/Output
//     PlcTask Inputs/GVL_iXlinker.EtherCAT_Master_EKxxxx.Beckhoff_EK18xx.Beckhoff_EK18xxEK1122.A_0004_EK1814_0000_0019.WcState.WcState <-> WcState/WcState
//     PlcTask Inputs/GVL_iXlinker.EtherCAT_Master_EKxxxx.Beckhoff_EK18xx.Beckhoff_EK18xxEK1122.A_0004_EK1814_0000_0019.WcState.InputToggle <-> WcState/InputToggle
//     PlcTask Inputs/GVL_iXlinker.EtherCAT_Master_EKxxxx.Beckhoff_EK18xx.Beckhoff_EK18xxEK1122.A_0004_EK1814_0000_0019.InfoData.State <-> InfoData/State
//   PLC/PLC Instance <-> EtherCAT Master EKxxxx/Beckhoff EK18xx/Beckhoff EK18xxEK1122/A_0005(EK1818-0000-0016)
//     PlcTask Inputs/GVL_iXlinker.EtherCAT_Master_EKxxxx.Beckhoff_EK18xx.Beckhoff_EK18xxEK1122.A_0005_EK1818_0000_0016.Channel_1.Input <-> Channel 1/Input
//     PlcTask Inputs/GVL_iXlinker.EtherCAT_Master_EKxxxx.Beckhoff_EK18xx.Beckhoff_EK18xxEK1122.A_0005_EK1818_0000_0016.Channel_2.Input <-> Channel 2/Input
//     PlcTask Inputs/GVL_iXlinker.EtherCAT_Master_EKxxxx.Beckhoff_EK18xx.Beckhoff_EK18xxEK1122.A_0005_EK1818_0000_0016.Channel_3.Input <-> Channel 3/Input
//     PlcTask Inputs/GVL_iXlinker.EtherCAT_Master_EKxxxx.Beckhoff_EK18xx.Beckhoff_EK18xxEK1122.A_0005_EK1818_0000_0016.Channel_4.Input <-> Channel 4/Input
//     PlcTask Inputs/GVL_iXlinker.EtherCAT_Master_EKxxxx.Beckhoff_EK18xx.Beckhoff_EK18xxEK1122.A_0005_EK1818_0000_0016.Channel_5.Input <-> Channel 5/Input
//     PlcTask Inputs/GVL_iXlinker.EtherCAT_Master_EKxxxx.Beckhoff_EK18xx.Beckhoff_EK18xxEK1122.A_0005_EK1818_0000_0016.Channel_6.Input <-> Channel 6/Input
//     PlcTask Inputs/GVL_iXlinker.EtherCAT_Master_EKxxxx.Beckhoff_EK18xx.Beckhoff_EK18xxEK1122.A_0005_EK1818_0000_0016.Channel_7.Input <-> Channel 7/Input
//     PlcTask Inputs/GVL_iXlinker.EtherCAT_Master_EKxxxx.Beckhoff_EK18xx.Beckhoff_EK18xxEK1122.A_0005_EK1818_0000_0016.Channel_8.Input <-> Channel 8/Input
//     PlcTask Outputs/GVL_iXlinker.EtherCAT_Master_EKxxxx.Beckhoff_EK18xx.Beckhoff_EK18xxEK1122.A_0005_EK1818_0000_0016.Channel_9.Output <-> Channel 9/Output
//     PlcTask Outputs/GVL_iXlinker.EtherCAT_Master_EKxxxx.Beckhoff_EK18xx.Beckhoff_EK18xxEK1122.A_0005_EK1818_0000_0016.Channel_10.Output <-> Channel 10/Output
//     PlcTask Outputs/GVL_iXlinker.EtherCAT_Master_EKxxxx.Beckhoff_EK18xx.Beckhoff_EK18xxEK1122.A_0005_EK1818_0000_0016.Channel_11.Output <-> Channel 11/Output
//     PlcTask Outputs/GVL_iXlinker.EtherCAT_Master_EKxxxx.Beckhoff_EK18xx.Beckhoff_EK18xxEK1122.A_0005_EK1818_0000_0016.Channel_12.Output <-> Channel 12/Output
//     PlcTask Inputs/GVL_iXlinker.EtherCAT_Master_EKxxxx.Beckhoff_EK18xx.Beckhoff_EK18xxEK1122.A_0005_EK1818_0000_0016.WcState.WcState <-> WcState/WcState
//     PlcTask Inputs/GVL_iXlinker.EtherCAT_Master_EKxxxx.Beckhoff_EK18xx.Beckhoff_EK18xxEK1122.A_0005_EK1818_0000_0016.WcState.InputToggle <-> WcState/InputToggle
//     PlcTask Inputs/GVL_iXlinker.EtherCAT_Master_EKxxxx.Beckhoff_EK18xx.Beckhoff_EK18xxEK1122.A_0005_EK1818_0000_0016.InfoData.State <-> InfoData/State
//   PLC/PLC Instance <-> EtherCAT Master EKxxxx/Beckhoff EK18xx/Beckhoff EK18xxEK1122/A_0006(EK1818-0000-0017)
//     PlcTask Inputs/GVL_iXlinker.EtherCAT_Master_EKxxxx.Beckhoff_EK18xx.Beckhoff_EK18xxEK1122.A_0006_EK1818_0000_0017.Channel_1.Input <-> Channel 1/Input
//     PlcTask Inputs/GVL_iXlinker.EtherCAT_Master_EKxxxx.Beckhoff_EK18xx.Beckhoff_EK18xxEK1122.A_0006_EK1818_0000_0017.Channel_2.Input <-> Channel 2/Input
//     PlcTask Inputs/GVL_iXlinker.EtherCAT_Master_EKxxxx.Beckhoff_EK18xx.Beckhoff_EK18xxEK1122.A_0006_EK1818_0000_0017.Channel_3.Input <-> Channel 3/Input
//     PlcTask Inputs/GVL_iXlinker.EtherCAT_Master_EKxxxx.Beckhoff_EK18xx.Beckhoff_EK18xxEK1122.A_0006_EK1818_0000_0017.Channel_4.Input <-> Channel 4/Input
//     PlcTask Inputs/GVL_iXlinker.EtherCAT_Master_EKxxxx.Beckhoff_EK18xx.Beckhoff_EK18xxEK1122.A_0006_EK1818_0000_0017.Channel_5.Input <-> Channel 5/Input
//     PlcTask Inputs/GVL_iXlinker.EtherCAT_Master_EKxxxx.Beckhoff_EK18xx.Beckhoff_EK18xxEK1122.A_0006_EK1818_0000_0017.Channel_6.Input <-> Channel 6/Input
//     PlcTask Inputs/GVL_iXlinker.EtherCAT_Master_EKxxxx.Beckhoff_EK18xx.Beckhoff_EK18xxEK1122.A_0006_EK1818_0000_0017.Channel_7.Input <-> Channel 7/Input
//     PlcTask Inputs/GVL_iXlinker.EtherCAT_Master_EKxxxx.Beckhoff_EK18xx.Beckhoff_EK18xxEK1122.A_0006_EK1818_0000_0017.Channel_8.Input <-> Channel 8/Input
//     PlcTask Outputs/GVL_iXlinker.EtherCAT_Master_EKxxxx.Beckhoff_EK18xx.Beckhoff_EK18xxEK1122.A_0006_EK1818_0000_0017.Channel_9.Output <-> Channel 9/Output
//     PlcTask Outputs/GVL_iXlinker.EtherCAT_Master_EKxxxx.Beckhoff_EK18xx.Beckhoff_EK18xxEK1122.A_0006_EK1818_0000_0017.Channel_10.Output <-> Channel 10/Output
//     PlcTask Outputs/GVL_iXlinker.EtherCAT_Master_EKxxxx.Beckhoff_EK18xx.Beckhoff_EK18xxEK1122.A_0006_EK1818_0000_0017.Channel_11.Output <-> Channel 11/Output
//     PlcTask Outputs/GVL_iXlinker.EtherCAT_Master_EKxxxx.Beckhoff_EK18xx.Beckhoff_EK18xxEK1122.A_0006_EK1818_0000_0017.Channel_12.Output <-> Channel 12/Output
//     PlcTask Inputs/GVL_iXlinker.EtherCAT_Master_EKxxxx.Beckhoff_EK18xx.Beckhoff_EK18xxEK1122.A_0006_EK1818_0000_0017.WcState.WcState <-> WcState/WcState
//     PlcTask Inputs/GVL_iXlinker.EtherCAT_Master_EKxxxx.Beckhoff_EK18xx.Beckhoff_EK18xxEK1122.A_0006_EK1818_0000_0017.WcState.InputToggle <-> WcState/InputToggle
//     PlcTask Inputs/GVL_iXlinker.EtherCAT_Master_EKxxxx.Beckhoff_EK18xx.Beckhoff_EK18xxEK1122.A_0006_EK1818_0000_0017.InfoData.State <-> InfoData/State
//   PLC/PLC Instance <-> EtherCAT Master EKxxxx/Beckhoff EK18xx/Beckhoff EK18xxEK1122/A_0007(EK1818-0000-0018)
//     PlcTask Inputs/GVL_iXlinker.EtherCAT_Master_EKxxxx.Beckhoff_EK18xx.Beckhoff_EK18xxEK1122.A_0007_EK1818_0000_0018.Channel_1.Input <-> Channel 1/Input
//     PlcTask Inputs/GVL_iXlinker.EtherCAT_Master_EKxxxx.Beckhoff_EK18xx.Beckhoff_EK18xxEK1122.A_0007_EK1818_0000_0018.Channel_2.Input <-> Channel 2/Input
//     PlcTask Inputs/GVL_iXlinker.EtherCAT_Master_EKxxxx.Beckhoff_EK18xx.Beckhoff_EK18xxEK1122.A_0007_EK1818_0000_0018.Channel_3.Input <-> Channel 3/Input
//     PlcTask Inputs/GVL_iXlinker.EtherCAT_Master_EKxxxx.Beckhoff_EK18xx.Beckhoff_EK18xxEK1122.A_0007_EK1818_0000_0018.Channel_4.Input <-> Channel 4/Input
//     PlcTask Inputs/GVL_iXlinker.EtherCAT_Master_EKxxxx.Beckhoff_EK18xx.Beckhoff_EK18xxEK1122.A_0007_EK1818_0000_0018.Channel_5.Input <-> Channel 5/Input
//     PlcTask Inputs/GVL_iXlinker.EtherCAT_Master_EKxxxx.Beckhoff_EK18xx.Beckhoff_EK18xxEK1122.A_0007_EK1818_0000_0018.Channel_6.Input <-> Channel 6/Input
//     PlcTask Inputs/GVL_iXlinker.EtherCAT_Master_EKxxxx.Beckhoff_EK18xx.Beckhoff_EK18xxEK1122.A_0007_EK1818_0000_0018.Channel_7.Input <-> Channel 7/Input
//     PlcTask Inputs/GVL_iXlinker.EtherCAT_Master_EKxxxx.Beckhoff_EK18xx.Beckhoff_EK18xxEK1122.A_0007_EK1818_0000_0018.Channel_8.Input <-> Channel 8/Input
//     PlcTask Outputs/GVL_iXlinker.EtherCAT_Master_EKxxxx.Beckhoff_EK18xx.Beckhoff_EK18xxEK1122.A_0007_EK1818_0000_0018.Channel_9.Output <-> Channel 9/Output
//     PlcTask Outputs/GVL_iXlinker.EtherCAT_Master_EKxxxx.Beckhoff_EK18xx.Beckhoff_EK18xxEK1122.A_0007_EK1818_0000_0018.Channel_10.Output <-> Channel 10/Output
//     PlcTask Outputs/GVL_iXlinker.EtherCAT_Master_EKxxxx.Beckhoff_EK18xx.Beckhoff_EK18xxEK1122.A_0007_EK1818_0000_0018.Channel_11.Output <-> Channel 11/Output
//     PlcTask Outputs/GVL_iXlinker.EtherCAT_Master_EKxxxx.Beckhoff_EK18xx.Beckhoff_EK18xxEK1122.A_0007_EK1818_0000_0018.Channel_12.Output <-> Channel 12/Output
//     PlcTask Inputs/GVL_iXlinker.EtherCAT_Master_EKxxxx.Beckhoff_EK18xx.Beckhoff_EK18xxEK1122.A_0007_EK1818_0000_0018.WcState.WcState <-> WcState/WcState
//     PlcTask Inputs/GVL_iXlinker.EtherCAT_Master_EKxxxx.Beckhoff_EK18xx.Beckhoff_EK18xxEK1122.A_0007_EK1818_0000_0018.WcState.InputToggle <-> WcState/InputToggle
//     PlcTask Inputs/GVL_iXlinker.EtherCAT_Master_EKxxxx.Beckhoff_EK18xx.Beckhoff_EK18xxEK1122.A_0007_EK1818_0000_0018.InfoData.State <-> InfoData/State
//   PLC/PLC Instance <-> EtherCAT Master EKxxxx/Beckhoff EK18xx/Beckhoff EK18xxEK1122/A_0008(EK1828-0000-0016)
//     PlcTask Inputs/GVL_iXlinker.EtherCAT_Master_EKxxxx.Beckhoff_EK18xx.Beckhoff_EK18xxEK1122.A_0008_EK1828_0000_0016.Channel_1.Input <-> Channel 1/Input
//     PlcTask Inputs/GVL_iXlinker.EtherCAT_Master_EKxxxx.Beckhoff_EK18xx.Beckhoff_EK18xxEK1122.A_0008_EK1828_0000_0016.Channel_2.Input <-> Channel 2/Input
//     PlcTask Inputs/GVL_iXlinker.EtherCAT_Master_EKxxxx.Beckhoff_EK18xx.Beckhoff_EK18xxEK1122.A_0008_EK1828_0000_0016.Channel_3.Input <-> Channel 3/Input
//     PlcTask Inputs/GVL_iXlinker.EtherCAT_Master_EKxxxx.Beckhoff_EK18xx.Beckhoff_EK18xxEK1122.A_0008_EK1828_0000_0016.Channel_4.Input <-> Channel 4/Input
//     PlcTask Outputs/GVL_iXlinker.EtherCAT_Master_EKxxxx.Beckhoff_EK18xx.Beckhoff_EK18xxEK1122.A_0008_EK1828_0000_0016.Channel_5.Output <-> Channel 5/Output
//     PlcTask Outputs/GVL_iXlinker.EtherCAT_Master_EKxxxx.Beckhoff_EK18xx.Beckhoff_EK18xxEK1122.A_0008_EK1828_0000_0016.Channel_6.Output <-> Channel 6/Output
//     PlcTask Outputs/GVL_iXlinker.EtherCAT_Master_EKxxxx.Beckhoff_EK18xx.Beckhoff_EK18xxEK1122.A_0008_EK1828_0000_0016.Channel_7.Output <-> Channel 7/Output
//     PlcTask Outputs/GVL_iXlinker.EtherCAT_Master_EKxxxx.Beckhoff_EK18xx.Beckhoff_EK18xxEK1122.A_0008_EK1828_0000_0016.Channel_8.Output <-> Channel 8/Output
//     PlcTask Outputs/GVL_iXlinker.EtherCAT_Master_EKxxxx.Beckhoff_EK18xx.Beckhoff_EK18xxEK1122.A_0008_EK1828_0000_0016.Channel_9.Output <-> Channel 9/Output
//     PlcTask Outputs/GVL_iXlinker.EtherCAT_Master_EKxxxx.Beckhoff_EK18xx.Beckhoff_EK18xxEK1122.A_0008_EK1828_0000_0016.Channel_10.Output <-> Channel 10/Output
//     PlcTask Outputs/GVL_iXlinker.EtherCAT_Master_EKxxxx.Beckhoff_EK18xx.Beckhoff_EK18xxEK1122.A_0008_EK1828_0000_0016.Channel_11.Output <-> Channel 11/Output
//     PlcTask Outputs/GVL_iXlinker.EtherCAT_Master_EKxxxx.Beckhoff_EK18xx.Beckhoff_EK18xxEK1122.A_0008_EK1828_0000_0016.Channel_12.Output <-> Channel 12/Output
//     PlcTask Inputs/GVL_iXlinker.EtherCAT_Master_EKxxxx.Beckhoff_EK18xx.Beckhoff_EK18xxEK1122.A_0008_EK1828_0000_0016.WcState.WcState <-> WcState/WcState
//     PlcTask Inputs/GVL_iXlinker.EtherCAT_Master_EKxxxx.Beckhoff_EK18xx.Beckhoff_EK18xxEK1122.A_0008_EK1828_0000_0016.WcState.InputToggle <-> WcState/InputToggle
//     PlcTask Inputs/GVL_iXlinker.EtherCAT_Master_EKxxxx.Beckhoff_EK18xx.Beckhoff_EK18xxEK1122.A_0008_EK1828_0000_0016.InfoData.State <-> InfoData/State
//   PLC/PLC Instance <-> EtherCAT Master EKxxxx/Beckhoff EK18xx/Beckhoff EK18xxEK1122/A_0009(EK1828-0000-0017)
//     PlcTask Inputs/GVL_iXlinker.EtherCAT_Master_EKxxxx.Beckhoff_EK18xx.Beckhoff_EK18xxEK1122.A_0009_EK1828_0000_0017.Channel_1.Input <-> Channel 1/Input
//     PlcTask Inputs/GVL_iXlinker.EtherCAT_Master_EKxxxx.Beckhoff_EK18xx.Beckhoff_EK18xxEK1122.A_0009_EK1828_0000_0017.Channel_2.Input <-> Channel 2/Input
//     PlcTask Inputs/GVL_iXlinker.EtherCAT_Master_EKxxxx.Beckhoff_EK18xx.Beckhoff_EK18xxEK1122.A_0009_EK1828_0000_0017.Channel_3.Input <-> Channel 3/Input
//     PlcTask Inputs/GVL_iXlinker.EtherCAT_Master_EKxxxx.Beckhoff_EK18xx.Beckhoff_EK18xxEK1122.A_0009_EK1828_0000_0017.Channel_4.Input <-> Channel 4/Input
//     PlcTask Outputs/GVL_iXlinker.EtherCAT_Master_EKxxxx.Beckhoff_EK18xx.Beckhoff_EK18xxEK1122.A_0009_EK1828_0000_0017.Channel_5.Output <-> Channel 5/Output
//     PlcTask Outputs/GVL_iXlinker.EtherCAT_Master_EKxxxx.Beckhoff_EK18xx.Beckhoff_EK18xxEK1122.A_0009_EK1828_0000_0017.Channel_6.Output <-> Channel 6/Output
//     PlcTask Outputs/GVL_iXlinker.EtherCAT_Master_EKxxxx.Beckhoff_EK18xx.Beckhoff_EK18xxEK1122.A_0009_EK1828_0000_0017.Channel_7.Output <-> Channel 7/Output
//     PlcTask Outputs/GVL_iXlinker.EtherCAT_Master_EKxxxx.Beckhoff_EK18xx.Beckhoff_EK18xxEK1122.A_0009_EK1828_0000_0017.Channel_8.Output <-> Channel 8/Output
//     PlcTask Outputs/GVL_iXlinker.EtherCAT_Master_EKxxxx.Beckhoff_EK18xx.Beckhoff_EK18xxEK1122.A_0009_EK1828_0000_0017.Channel_9.Output <-> Channel 9/Output
//     PlcTask Outputs/GVL_iXlinker.EtherCAT_Master_EKxxxx.Beckhoff_EK18xx.Beckhoff_EK18xxEK1122.A_0009_EK1828_0000_0017.Channel_10.Output <-> Channel 10/Output
//     PlcTask Outputs/GVL_iXlinker.EtherCAT_Master_EKxxxx.Beckhoff_EK18xx.Beckhoff_EK18xxEK1122.A_0009_EK1828_0000_0017.Channel_11.Output <-> Channel 11/Output
//     PlcTask Outputs/GVL_iXlinker.EtherCAT_Master_EKxxxx.Beckhoff_EK18xx.Beckhoff_EK18xxEK1122.A_0009_EK1828_0000_0017.Channel_12.Output <-> Channel 12/Output
//     PlcTask Inputs/GVL_iXlinker.EtherCAT_Master_EKxxxx.Beckhoff_EK18xx.Beckhoff_EK18xxEK1122.A_0009_EK1828_0000_0017.WcState.WcState <-> WcState/WcState
//     PlcTask Inputs/GVL_iXlinker.EtherCAT_Master_EKxxxx.Beckhoff_EK18xx.Beckhoff_EK18xxEK1122.A_0009_EK1828_0000_0017.WcState.InputToggle <-> WcState/InputToggle
//     PlcTask Inputs/GVL_iXlinker.EtherCAT_Master_EKxxxx.Beckhoff_EK18xx.Beckhoff_EK18xxEK1122.A_0009_EK1828_0000_0017.InfoData.State <-> InfoData/State
//   PLC/PLC Instance <-> EtherCAT Master EKxxxx/Beckhoff EK18xx/Beckhoff EK18xxEK1122/A_0010(EK1828-0000-0018)
//     PlcTask Inputs/GVL_iXlinker.EtherCAT_Master_EKxxxx.Beckhoff_EK18xx.Beckhoff_EK18xxEK1122.A_0010_EK1828_0000_0018.Channel_1.Input <-> Channel 1/Input
//     PlcTask Inputs/GVL_iXlinker.EtherCAT_Master_EKxxxx.Beckhoff_EK18xx.Beckhoff_EK18xxEK1122.A_0010_EK1828_0000_0018.Channel_2.Input <-> Channel 2/Input
//     PlcTask Inputs/GVL_iXlinker.EtherCAT_Master_EKxxxx.Beckhoff_EK18xx.Beckhoff_EK18xxEK1122.A_0010_EK1828_0000_0018.Channel_3.Input <-> Channel 3/Input
//     PlcTask Inputs/GVL_iXlinker.EtherCAT_Master_EKxxxx.Beckhoff_EK18xx.Beckhoff_EK18xxEK1122.A_0010_EK1828_0000_0018.Channel_4.Input <-> Channel 4/Input
//     PlcTask Outputs/GVL_iXlinker.EtherCAT_Master_EKxxxx.Beckhoff_EK18xx.Beckhoff_EK18xxEK1122.A_0010_EK1828_0000_0018.Channel_5.Output <-> Channel 5/Output
//     PlcTask Outputs/GVL_iXlinker.EtherCAT_Master_EKxxxx.Beckhoff_EK18xx.Beckhoff_EK18xxEK1122.A_0010_EK1828_0000_0018.Channel_6.Output <-> Channel 6/Output
//     PlcTask Outputs/GVL_iXlinker.EtherCAT_Master_EKxxxx.Beckhoff_EK18xx.Beckhoff_EK18xxEK1122.A_0010_EK1828_0000_0018.Channel_7.Output <-> Channel 7/Output
//     PlcTask Outputs/GVL_iXlinker.EtherCAT_Master_EKxxxx.Beckhoff_EK18xx.Beckhoff_EK18xxEK1122.A_0010_EK1828_0000_0018.Channel_8.Output <-> Channel 8/Output
//     PlcTask Outputs/GVL_iXlinker.EtherCAT_Master_EKxxxx.Beckhoff_EK18xx.Beckhoff_EK18xxEK1122.A_0010_EK1828_0000_0018.Channel_9.Output <-> Channel 9/Output
//     PlcTask Outputs/GVL_iXlinker.EtherCAT_Master_EKxxxx.Beckhoff_EK18xx.Beckhoff_EK18xxEK1122.A_0010_EK1828_0000_0018.Channel_10.Output <-> Channel 10/Output
//     PlcTask Outputs/GVL_iXlinker.EtherCAT_Master_EKxxxx.Beckhoff_EK18xx.Beckhoff_EK18xxEK1122.A_0010_EK1828_0000_0018.Channel_11.Output <-> Channel 11/Output
//     PlcTask Outputs/GVL_iXlinker.EtherCAT_Master_EKxxxx.Beckhoff_EK18xx.Beckhoff_EK18xxEK1122.A_0010_EK1828_0000_0018.Channel_12.Output <-> Channel 12/Output
//     PlcTask Inputs/GVL_iXlinker.EtherCAT_Master_EKxxxx.Beckhoff_EK18xx.Beckhoff_EK18xxEK1122.A_0010_EK1828_0000_0018.WcState.WcState <-> WcState/WcState
//     PlcTask Inputs/GVL_iXlinker.EtherCAT_Master_EKxxxx.Beckhoff_EK18xx.Beckhoff_EK18xxEK1122.A_0010_EK1828_0000_0018.WcState.InputToggle <-> WcState/InputToggle
//     PlcTask Inputs/GVL_iXlinker.EtherCAT_Master_EKxxxx.Beckhoff_EK18xx.Beckhoff_EK18xxEK1122.A_0010_EK1828_0000_0018.InfoData.State <-> InfoData/State
//   PLC/PLC Instance <-> EtherCAT Master EKxxxx/Beckhoff EK18xx/Beckhoff EK18xxEK1122/A_0011(EK1828-0010-0016)
//     PlcTask Outputs/GVL_iXlinker.EtherCAT_Master_EKxxxx.Beckhoff_EK18xx.Beckhoff_EK18xxEK1122.A_0011_EK1828_0010_0016.Channel_1.Output <-> Channel 1/Output
//     PlcTask Outputs/GVL_iXlinker.EtherCAT_Master_EKxxxx.Beckhoff_EK18xx.Beckhoff_EK18xxEK1122.A_0011_EK1828_0010_0016.Channel_2.Output <-> Channel 2/Output
//     PlcTask Outputs/GVL_iXlinker.EtherCAT_Master_EKxxxx.Beckhoff_EK18xx.Beckhoff_EK18xxEK1122.A_0011_EK1828_0010_0016.Channel_3.Output <-> Channel 3/Output
//     PlcTask Outputs/GVL_iXlinker.EtherCAT_Master_EKxxxx.Beckhoff_EK18xx.Beckhoff_EK18xxEK1122.A_0011_EK1828_0010_0016.Channel_4.Output <-> Channel 4/Output
//     PlcTask Outputs/GVL_iXlinker.EtherCAT_Master_EKxxxx.Beckhoff_EK18xx.Beckhoff_EK18xxEK1122.A_0011_EK1828_0010_0016.Channel_5.Output <-> Channel 5/Output
//     PlcTask Outputs/GVL_iXlinker.EtherCAT_Master_EKxxxx.Beckhoff_EK18xx.Beckhoff_EK18xxEK1122.A_0011_EK1828_0010_0016.Channel_6.Output <-> Channel 6/Output
//     PlcTask Outputs/GVL_iXlinker.EtherCAT_Master_EKxxxx.Beckhoff_EK18xx.Beckhoff_EK18xxEK1122.A_0011_EK1828_0010_0016.Channel_7.Output <-> Channel 7/Output
//     PlcTask Outputs/GVL_iXlinker.EtherCAT_Master_EKxxxx.Beckhoff_EK18xx.Beckhoff_EK18xxEK1122.A_0011_EK1828_0010_0016.Channel_8.Output <-> Channel 8/Output
//     PlcTask Inputs/GVL_iXlinker.EtherCAT_Master_EKxxxx.Beckhoff_EK18xx.Beckhoff_EK18xxEK1122.A_0011_EK1828_0010_0016.WcState.WcState <-> WcState/WcState
//     PlcTask Inputs/GVL_iXlinker.EtherCAT_Master_EKxxxx.Beckhoff_EK18xx.Beckhoff_EK18xxEK1122.A_0011_EK1828_0010_0016.InfoData.State <-> InfoData/State
//   PLC/PLC Instance <-> EtherCAT Master EKxxxx/Beckhoff EK18xx/Beckhoff EK18xxEK1122/A_0012(EK1828-0010-0017)
//     PlcTask Outputs/GVL_iXlinker.EtherCAT_Master_EKxxxx.Beckhoff_EK18xx.Beckhoff_EK18xxEK1122.A_0012_EK1828_0010_0017.Channel_1.Output <-> Channel 1/Output
//     PlcTask Outputs/GVL_iXlinker.EtherCAT_Master_EKxxxx.Beckhoff_EK18xx.Beckhoff_EK18xxEK1122.A_0012_EK1828_0010_0017.Channel_2.Output <-> Channel 2/Output
//     PlcTask Outputs/GVL_iXlinker.EtherCAT_Master_EKxxxx.Beckhoff_EK18xx.Beckhoff_EK18xxEK1122.A_0012_EK1828_0010_0017.Channel_3.Output <-> Channel 3/Output
//     PlcTask Outputs/GVL_iXlinker.EtherCAT_Master_EKxxxx.Beckhoff_EK18xx.Beckhoff_EK18xxEK1122.A_0012_EK1828_0010_0017.Channel_4.Output <-> Channel 4/Output
//     PlcTask Outputs/GVL_iXlinker.EtherCAT_Master_EKxxxx.Beckhoff_EK18xx.Beckhoff_EK18xxEK1122.A_0012_EK1828_0010_0017.Channel_5.Output <-> Channel 5/Output
//     PlcTask Outputs/GVL_iXlinker.EtherCAT_Master_EKxxxx.Beckhoff_EK18xx.Beckhoff_EK18xxEK1122.A_0012_EK1828_0010_0017.Channel_6.Output <-> Channel 6/Output
//     PlcTask Outputs/GVL_iXlinker.EtherCAT_Master_EKxxxx.Beckhoff_EK18xx.Beckhoff_EK18xxEK1122.A_0012_EK1828_0010_0017.Channel_7.Output <-> Channel 7/Output
//     PlcTask Outputs/GVL_iXlinker.EtherCAT_Master_EKxxxx.Beckhoff_EK18xx.Beckhoff_EK18xxEK1122.A_0012_EK1828_0010_0017.Channel_8.Output <-> Channel 8/Output
//     PlcTask Inputs/GVL_iXlinker.EtherCAT_Master_EKxxxx.Beckhoff_EK18xx.Beckhoff_EK18xxEK1122.A_0012_EK1828_0010_0017.WcState.WcState <-> WcState/WcState
//     PlcTask Inputs/GVL_iXlinker.EtherCAT_Master_EKxxxx.Beckhoff_EK18xx.Beckhoff_EK18xxEK1122.A_0012_EK1828_0010_0017.InfoData.State <-> InfoData/State
//   PLC/PLC Instance <-> EtherCAT Master EKxxxx/Beckhoff EK18xx/Beckhoff EK18xxEK1122/A_0013(EK1828-0010-0018)
//     PlcTask Outputs/GVL_iXlinker.EtherCAT_Master_EKxxxx.Beckhoff_EK18xx.Beckhoff_EK18xxEK1122.A_0013_EK1828_0010_0018.Channel_1.Output <-> Channel 1/Output
//     PlcTask Outputs/GVL_iXlinker.EtherCAT_Master_EKxxxx.Beckhoff_EK18xx.Beckhoff_EK18xxEK1122.A_0013_EK1828_0010_0018.Channel_2.Output <-> Channel 2/Output
//     PlcTask Outputs/GVL_iXlinker.EtherCAT_Master_EKxxxx.Beckhoff_EK18xx.Beckhoff_EK18xxEK1122.A_0013_EK1828_0010_0018.Channel_3.Output <-> Channel 3/Output
//     PlcTask Outputs/GVL_iXlinker.EtherCAT_Master_EKxxxx.Beckhoff_EK18xx.Beckhoff_EK18xxEK1122.A_0013_EK1828_0010_0018.Channel_4.Output <-> Channel 4/Output
//     PlcTask Outputs/GVL_iXlinker.EtherCAT_Master_EKxxxx.Beckhoff_EK18xx.Beckhoff_EK18xxEK1122.A_0013_EK1828_0010_0018.Channel_5.Output <-> Channel 5/Output
//     PlcTask Outputs/GVL_iXlinker.EtherCAT_Master_EKxxxx.Beckhoff_EK18xx.Beckhoff_EK18xxEK1122.A_0013_EK1828_0010_0018.Channel_6.Output <-> Channel 6/Output
//     PlcTask Outputs/GVL_iXlinker.EtherCAT_Master_EKxxxx.Beckhoff_EK18xx.Beckhoff_EK18xxEK1122.A_0013_EK1828_0010_0018.Channel_7.Output <-> Channel 7/Output
//     PlcTask Outputs/GVL_iXlinker.EtherCAT_Master_EKxxxx.Beckhoff_EK18xx.Beckhoff_EK18xxEK1122.A_0013_EK1828_0010_0018.Channel_8.Output <-> Channel 8/Output
//     PlcTask Inputs/GVL_iXlinker.EtherCAT_Master_EKxxxx.Beckhoff_EK18xx.Beckhoff_EK18xxEK1122.A_0013_EK1828_0010_0018.WcState.WcState <-> WcState/WcState
//     PlcTask Inputs/GVL_iXlinker.EtherCAT_Master_EKxxxx.Beckhoff_EK18xx.Beckhoff_EK18xxEK1122.A_0013_EK1828_0010_0018.InfoData.State <-> InfoData/State
//   PLC/PLC Instance <-> EtherCAT Master EKxxxx/Beckhoff EKM1xxx
//     PlcTask Inputs/GVL_iXlinker.EtherCAT_Master_EKxxxx.Beckhoff_EKM1xxx.InfoData.State <-> InfoData/State
//   PLC/PLC Instance <-> EtherCAT Master EKxxxx/Beckhoff EKM1xxx/Beckhoff EKM1xxxEK1122
//     PlcTask Inputs/GVL_iXlinker.EtherCAT_Master_EKxxxx.Beckhoff_EKM1xxx.Beckhoff_EKM1xxxEK1122.InfoData.State <-> InfoData/State
//   PLC/PLC Instance <-> EtherCAT Master EKxxxx/Beckhoff EKM1xxx/Beckhoff EKM1xxxEK1122/Beckhoff EKM1xxxsub EK1100
//     PlcTask Inputs/GVL_iXlinker.EtherCAT_Master_EKxxxx.Beckhoff_EKM1xxx.Beckhoff_EKM1xxxEK1122.Beckhoff_EKM1xxxsub_EK1100.InfoData.State <-> InfoData/State
//   PLC/PLC Instance <-> EtherCAT Master EKxxxx/Beckhoff EKM1xxx/Beckhoff EKM1xxxEK1122/A_0001(EKM1101-0000-0016)
//     PlcTask Inputs/GVL_iXlinker.EtherCAT_Master_EKxxxx.Beckhoff_EKM1xxx.Beckhoff_EKM1xxxEK1122.A_0001_EKM1101_0000_0016.MMS_Device_Inputs.Status/Diag <-> MMS Device Inputs/Status/Diag
//     PlcTask Inputs/GVL_iXlinker.EtherCAT_Master_EKxxxx.Beckhoff_EKM1xxx.Beckhoff_EKM1xxxEK1122.A_0001_EKM1101_0000_0016.MMS_Device_Inputs.Status/Error <-> MMS Device Inputs/Status/Error
//     PlcTask Inputs/GVL_iXlinker.EtherCAT_Master_EKxxxx.Beckhoff_EKM1xxx.Beckhoff_EKM1xxxEK1122.A_0001_EKM1101_0000_0016.MMS_Device_Inputs.Status/Input_cycle_Counter <-> MMS Device Inputs/Status/Input cycle Counter
//     PlcTask Inputs/GVL_iXlinker.EtherCAT_Master_EKxxxx.Beckhoff_EKM1xxx.Beckhoff_EKM1xxxEK1122.A_0001_EKM1101_0000_0016.MMS_Device_Inputs.Status/TxPDO_State <-> MMS Device Inputs/Status/TxPDO State
//     PlcTask Inputs/GVL_iXlinker.EtherCAT_Master_EKxxxx.Beckhoff_EKM1xxx.Beckhoff_EKM1xxxEK1122.A_0001_EKM1101_0000_0016.MMS_Device_Inputs.Status/ID <-> MMS Device Inputs/Status/ID
//     PlcTask Inputs/GVL_iXlinker.EtherCAT_Master_EKxxxx.Beckhoff_EKM1xxx.Beckhoff_EKM1xxxEK1122.A_0001_EKM1101_0000_0016.MMS_Acceleration_Status.Status/Error <-> MMS Acceleration Status/Status/Error
//     PlcTask Inputs/GVL_iXlinker.EtherCAT_Master_EKxxxx.Beckhoff_EKM1xxx.Beckhoff_EKM1xxxEK1122.A_0001_EKM1101_0000_0016.MMS_Acceleration_Status.Status/Underrange <-> MMS Acceleration Status/Status/Underrange
//     PlcTask Inputs/GVL_iXlinker.EtherCAT_Master_EKxxxx.Beckhoff_EKM1xxx.Beckhoff_EKM1xxxEK1122.A_0001_EKM1101_0000_0016.MMS_Acceleration_Status.Status/Overrange <-> MMS Acceleration Status/Status/Overrange
//     PlcTask Inputs/GVL_iXlinker.EtherCAT_Master_EKxxxx.Beckhoff_EKM1xxx.Beckhoff_EKM1xxxEK1122.A_0001_EKM1101_0000_0016.MMS_Acceleration_Status.Status/Diag <-> MMS Acceleration Status/Status/Diag
//     PlcTask Inputs/GVL_iXlinker.EtherCAT_Master_EKxxxx.Beckhoff_EKM1xxx.Beckhoff_EKM1xxxEK1122.A_0001_EKM1101_0000_0016.MMS_Acceleration_Status.Status/Sensor_Ovr <-> MMS Acceleration Status/Status/Sensor Ovr
//     PlcTask Inputs/GVL_iXlinker.EtherCAT_Master_EKxxxx.Beckhoff_EKM1xxx.Beckhoff_EKM1xxxEK1122.A_0001_EKM1101_0000_0016.MMS_Acceleration_Status.Status/Overrun <-> MMS Acceleration Status/Status/Overrun
//     PlcTask Inputs/GVL_iXlinker.EtherCAT_Master_EKxxxx.Beckhoff_EKM1xxx.Beckhoff_EKM1xxxEK1122.A_0001_EKM1101_0000_0016.MMS_Acceleration_Status.Status/TxPDO_State <-> MMS Acceleration Status/Status/TxPDO State
//     PlcTask Inputs/GVL_iXlinker.EtherCAT_Master_EKxxxx.Beckhoff_EKM1xxx.Beckhoff_EKM1xxxEK1122.A_0001_EKM1101_0000_0016.MMS_Acceleration_Status.Number_of_samples <-> MMS Acceleration Status/Number of samples
//     PlcTask Inputs/GVL_iXlinker.EtherCAT_Master_EKxxxx.Beckhoff_EKM1xxx.Beckhoff_EKM1xxxEK1122.A_0001_EKM1101_0000_0016.MMS_Acceleration_X_Axis.Value <-> MMS Acceleration X-Axis/Value
//     PlcTask Inputs/GVL_iXlinker.EtherCAT_Master_EKxxxx.Beckhoff_EKM1xxx.Beckhoff_EKM1xxxEK1122.A_0001_EKM1101_0000_0016.MMS_Acceleration_Y_Axis.Value <-> MMS Acceleration Y-Axis/Value
//     PlcTask Inputs/GVL_iXlinker.EtherCAT_Master_EKxxxx.Beckhoff_EKM1xxx.Beckhoff_EKM1xxxEK1122.A_0001_EKM1101_0000_0016.MMS_Acceleration_Z_Axis.Value <-> MMS Acceleration Z-Axis/Value
//     PlcTask Inputs/GVL_iXlinker.EtherCAT_Master_EKxxxx.Beckhoff_EKM1xxx.Beckhoff_EKM1xxxEK1122.A_0001_EKM1101_0000_0016.MMS_Acceleration_Timestamp.Timestamp <-> MMS Acceleration Timestamp/Timestamp
//     PlcTask Inputs/GVL_iXlinker.EtherCAT_Master_EKxxxx.Beckhoff_EKM1xxx.Beckhoff_EKM1xxxEK1122.A_0001_EKM1101_0000_0016.MMS_Voltage_Us_In_Inputs.Status/Underrange <-> MMS Voltage Us In Inputs/Status/Underrange
//     PlcTask Inputs/GVL_iXlinker.EtherCAT_Master_EKxxxx.Beckhoff_EKM1xxx.Beckhoff_EKM1xxxEK1122.A_0001_EKM1101_0000_0016.MMS_Voltage_Us_In_Inputs.Status/Overrange <-> MMS Voltage Us In Inputs/Status/Overrange
//     PlcTask Inputs/GVL_iXlinker.EtherCAT_Master_EKxxxx.Beckhoff_EKM1xxx.Beckhoff_EKM1xxxEK1122.A_0001_EKM1101_0000_0016.MMS_Voltage_Us_In_Inputs.Status/Limit_1 <-> MMS Voltage Us In Inputs/Status/Limit 1
//     PlcTask Inputs/GVL_iXlinker.EtherCAT_Master_EKxxxx.Beckhoff_EKM1xxx.Beckhoff_EKM1xxxEK1122.A_0001_EKM1101_0000_0016.MMS_Voltage_Us_In_Inputs.Status/Limit_2 <-> MMS Voltage Us In Inputs/Status/Limit 2
//     PlcTask Inputs/GVL_iXlinker.EtherCAT_Master_EKxxxx.Beckhoff_EKM1xxx.Beckhoff_EKM1xxxEK1122.A_0001_EKM1101_0000_0016.MMS_Voltage_Us_In_Inputs.Status/Error <-> MMS Voltage Us In Inputs/Status/Error
//     PlcTask Inputs/GVL_iXlinker.EtherCAT_Master_EKxxxx.Beckhoff_EKM1xxx.Beckhoff_EKM1xxxEK1122.A_0001_EKM1101_0000_0016.MMS_Voltage_Us_In_Inputs.Status/TxPDO_State <-> MMS Voltage Us In Inputs/Status/TxPDO State
//     PlcTask Inputs/GVL_iXlinker.EtherCAT_Master_EKxxxx.Beckhoff_EKM1xxx.Beckhoff_EKM1xxxEK1122.A_0001_EKM1101_0000_0016.MMS_Voltage_Us_In_Inputs.Status/TxPDO_Toggle <-> MMS Voltage Us In Inputs/Status/TxPDO Toggle
//     PlcTask Inputs/GVL_iXlinker.EtherCAT_Master_EKxxxx.Beckhoff_EKM1xxx.Beckhoff_EKM1xxxEK1122.A_0001_EKM1101_0000_0016.MMS_Voltage_Us_In_Inputs.Value <-> MMS Voltage Us In Inputs/Value
//     PlcTask Inputs/GVL_iXlinker.EtherCAT_Master_EKxxxx.Beckhoff_EKM1xxx.Beckhoff_EKM1xxxEK1122.A_0001_EKM1101_0000_0016.MMS_Voltage_Up_In_Inputs.Status/Underrange <-> MMS Voltage Up In Inputs/Status/Underrange
//     PlcTask Inputs/GVL_iXlinker.EtherCAT_Master_EKxxxx.Beckhoff_EKM1xxx.Beckhoff_EKM1xxxEK1122.A_0001_EKM1101_0000_0016.MMS_Voltage_Up_In_Inputs.Status/Overrange <-> MMS Voltage Up In Inputs/Status/Overrange
//     PlcTask Inputs/GVL_iXlinker.EtherCAT_Master_EKxxxx.Beckhoff_EKM1xxx.Beckhoff_EKM1xxxEK1122.A_0001_EKM1101_0000_0016.MMS_Voltage_Up_In_Inputs.Status/Limit_1 <-> MMS Voltage Up In Inputs/Status/Limit 1
//     PlcTask Inputs/GVL_iXlinker.EtherCAT_Master_EKxxxx.Beckhoff_EKM1xxx.Beckhoff_EKM1xxxEK1122.A_0001_EKM1101_0000_0016.MMS_Voltage_Up_In_Inputs.Status/Limit_2 <-> MMS Voltage Up In Inputs/Status/Limit 2
//     PlcTask Inputs/GVL_iXlinker.EtherCAT_Master_EKxxxx.Beckhoff_EKM1xxx.Beckhoff_EKM1xxxEK1122.A_0001_EKM1101_0000_0016.MMS_Voltage_Up_In_Inputs.Status/Error <-> MMS Voltage Up In Inputs/Status/Error
//     PlcTask Inputs/GVL_iXlinker.EtherCAT_Master_EKxxxx.Beckhoff_EKM1xxx.Beckhoff_EKM1xxxEK1122.A_0001_EKM1101_0000_0016.MMS_Voltage_Up_In_Inputs.Status/TxPDO_State <-> MMS Voltage Up In Inputs/Status/TxPDO State
//     PlcTask Inputs/GVL_iXlinker.EtherCAT_Master_EKxxxx.Beckhoff_EKM1xxx.Beckhoff_EKM1xxxEK1122.A_0001_EKM1101_0000_0016.MMS_Voltage_Up_In_Inputs.Status/TxPDO_Toggle <-> MMS Voltage Up In Inputs/Status/TxPDO Toggle
//     PlcTask Inputs/GVL_iXlinker.EtherCAT_Master_EKxxxx.Beckhoff_EKM1xxx.Beckhoff_EKM1xxxEK1122.A_0001_EKM1101_0000_0016.MMS_Voltage_Up_In_Inputs.Value <-> MMS Voltage Up In Inputs/Value
//     PlcTask Inputs/GVL_iXlinker.EtherCAT_Master_EKxxxx.Beckhoff_EKM1xxx.Beckhoff_EKM1xxxEK1122.A_0001_EKM1101_0000_0016.MMS_Voltage_Up_Out_Inputs.Status/Underrange <-> MMS Voltage Up Out Inputs/Status/Underrange
//     PlcTask Inputs/GVL_iXlinker.EtherCAT_Master_EKxxxx.Beckhoff_EKM1xxx.Beckhoff_EKM1xxxEK1122.A_0001_EKM1101_0000_0016.MMS_Voltage_Up_Out_Inputs.Status/Overrange <-> MMS Voltage Up Out Inputs/Status/Overrange
//     PlcTask Inputs/GVL_iXlinker.EtherCAT_Master_EKxxxx.Beckhoff_EKM1xxx.Beckhoff_EKM1xxxEK1122.A_0001_EKM1101_0000_0016.MMS_Voltage_Up_Out_Inputs.Status/Limit_1 <-> MMS Voltage Up Out Inputs/Status/Limit 1
//     PlcTask Inputs/GVL_iXlinker.EtherCAT_Master_EKxxxx.Beckhoff_EKM1xxx.Beckhoff_EKM1xxxEK1122.A_0001_EKM1101_0000_0016.MMS_Voltage_Up_Out_Inputs.Status/Limit_2 <-> MMS Voltage Up Out Inputs/Status/Limit 2
//     PlcTask Inputs/GVL_iXlinker.EtherCAT_Master_EKxxxx.Beckhoff_EKM1xxx.Beckhoff_EKM1xxxEK1122.A_0001_EKM1101_0000_0016.MMS_Voltage_Up_Out_Inputs.Status/Error <-> MMS Voltage Up Out Inputs/Status/Error
//     PlcTask Inputs/GVL_iXlinker.EtherCAT_Master_EKxxxx.Beckhoff_EKM1xxx.Beckhoff_EKM1xxxEK1122.A_0001_EKM1101_0000_0016.MMS_Voltage_Up_Out_Inputs.Status/TxPDO_State <-> MMS Voltage Up Out Inputs/Status/TxPDO State
//     PlcTask Inputs/GVL_iXlinker.EtherCAT_Master_EKxxxx.Beckhoff_EKM1xxx.Beckhoff_EKM1xxxEK1122.A_0001_EKM1101_0000_0016.MMS_Voltage_Up_Out_Inputs.Status/TxPDO_Toggle <-> MMS Voltage Up Out Inputs/Status/TxPDO Toggle
//     PlcTask Inputs/GVL_iXlinker.EtherCAT_Master_EKxxxx.Beckhoff_EKM1xxx.Beckhoff_EKM1xxxEK1122.A_0001_EKM1101_0000_0016.MMS_Voltage_Up_Out_Inputs.Value <-> MMS Voltage Up Out Inputs/Value
//     PlcTask Outputs/GVL_iXlinker.EtherCAT_Master_EKxxxx.Beckhoff_EKM1xxx.Beckhoff_EKM1xxxEK1122.A_0001_EKM1101_0000_0016.MMS_Device_Outputs.Control/Up_Out_OFF <-> MMS Device Outputs/Control/Up Out OFF
//     PlcTask Inputs/GVL_iXlinker.EtherCAT_Master_EKxxxx.Beckhoff_EKM1xxx.Beckhoff_EKM1xxxEK1122.A_0001_EKM1101_0000_0016.WcState.WcState <-> WcState/WcState
//     PlcTask Inputs/GVL_iXlinker.EtherCAT_Master_EKxxxx.Beckhoff_EKM1xxx.Beckhoff_EKM1xxxEK1122.A_0001_EKM1101_0000_0016.WcState.InputToggle <-> WcState/InputToggle
//     PlcTask Inputs/GVL_iXlinker.EtherCAT_Master_EKxxxx.Beckhoff_EKM1xxx.Beckhoff_EKM1xxxEK1122.A_0001_EKM1101_0000_0016.InfoData.AdsAddr <-> InfoData/AdsAddr
//     PlcTask Inputs/GVL_iXlinker.EtherCAT_Master_EKxxxx.Beckhoff_EKM1xxx.Beckhoff_EKM1xxxEK1122.A_0001_EKM1101_0000_0016.InfoData.DcOutputShift <-> InfoData/DcOutputShift
//     PlcTask Inputs/GVL_iXlinker.EtherCAT_Master_EKxxxx.Beckhoff_EKM1xxx.Beckhoff_EKM1xxxEK1122.A_0001_EKM1101_0000_0016.InfoData.DcInputShift <-> InfoData/DcInputShift
//     PlcTask Inputs/GVL_iXlinker.EtherCAT_Master_EKxxxx.Beckhoff_EKM1xxx.Beckhoff_EKM1xxxEK1122.A_0001_EKM1101_0000_0016.InfoData.State <-> InfoData/State
//   PLC/PLC Instance <-> EtherCAT Master EKxxxx/Beckhoff EKM1xxx/Beckhoff EKM1xxxEK1122/A_0002(EKM1101-0000-0017)
//     PlcTask Inputs/GVL_iXlinker.EtherCAT_Master_EKxxxx.Beckhoff_EKM1xxx.Beckhoff_EKM1xxxEK1122.A_0002_EKM1101_0000_0017.MMS_Device_Inputs.Status/Diag <-> MMS Device Inputs/Status/Diag
//     PlcTask Inputs/GVL_iXlinker.EtherCAT_Master_EKxxxx.Beckhoff_EKM1xxx.Beckhoff_EKM1xxxEK1122.A_0002_EKM1101_0000_0017.MMS_Device_Inputs.Status/Error <-> MMS Device Inputs/Status/Error
//     PlcTask Inputs/GVL_iXlinker.EtherCAT_Master_EKxxxx.Beckhoff_EKM1xxx.Beckhoff_EKM1xxxEK1122.A_0002_EKM1101_0000_0017.MMS_Device_Inputs.Status/Input_cycle_Counter <-> MMS Device Inputs/Status/Input cycle Counter
//     PlcTask Inputs/GVL_iXlinker.EtherCAT_Master_EKxxxx.Beckhoff_EKM1xxx.Beckhoff_EKM1xxxEK1122.A_0002_EKM1101_0000_0017.MMS_Device_Inputs.Status/TxPDO_State <-> MMS Device Inputs/Status/TxPDO State
//     PlcTask Inputs/GVL_iXlinker.EtherCAT_Master_EKxxxx.Beckhoff_EKM1xxx.Beckhoff_EKM1xxxEK1122.A_0002_EKM1101_0000_0017.MMS_Device_Inputs.Status/ID <-> MMS Device Inputs/Status/ID
//     PlcTask Inputs/GVL_iXlinker.EtherCAT_Master_EKxxxx.Beckhoff_EKM1xxx.Beckhoff_EKM1xxxEK1122.A_0002_EKM1101_0000_0017.MMS_Acceleration_Status.Status/Error <-> MMS Acceleration Status/Status/Error
//     PlcTask Inputs/GVL_iXlinker.EtherCAT_Master_EKxxxx.Beckhoff_EKM1xxx.Beckhoff_EKM1xxxEK1122.A_0002_EKM1101_0000_0017.MMS_Acceleration_Status.Status/Underrange <-> MMS Acceleration Status/Status/Underrange
//     PlcTask Inputs/GVL_iXlinker.EtherCAT_Master_EKxxxx.Beckhoff_EKM1xxx.Beckhoff_EKM1xxxEK1122.A_0002_EKM1101_0000_0017.MMS_Acceleration_Status.Status/Overrange <-> MMS Acceleration Status/Status/Overrange
//     PlcTask Inputs/GVL_iXlinker.EtherCAT_Master_EKxxxx.Beckhoff_EKM1xxx.Beckhoff_EKM1xxxEK1122.A_0002_EKM1101_0000_0017.MMS_Acceleration_Status.Status/Diag <-> MMS Acceleration Status/Status/Diag
//     PlcTask Inputs/GVL_iXlinker.EtherCAT_Master_EKxxxx.Beckhoff_EKM1xxx.Beckhoff_EKM1xxxEK1122.A_0002_EKM1101_0000_0017.MMS_Acceleration_Status.Status/Sensor_Ovr <-> MMS Acceleration Status/Status/Sensor Ovr
//     PlcTask Inputs/GVL_iXlinker.EtherCAT_Master_EKxxxx.Beckhoff_EKM1xxx.Beckhoff_EKM1xxxEK1122.A_0002_EKM1101_0000_0017.MMS_Acceleration_Status.Status/Overrun <-> MMS Acceleration Status/Status/Overrun
//     PlcTask Inputs/GVL_iXlinker.EtherCAT_Master_EKxxxx.Beckhoff_EKM1xxx.Beckhoff_EKM1xxxEK1122.A_0002_EKM1101_0000_0017.MMS_Acceleration_Status.Status/TxPDO_State <-> MMS Acceleration Status/Status/TxPDO State
//     PlcTask Inputs/GVL_iXlinker.EtherCAT_Master_EKxxxx.Beckhoff_EKM1xxx.Beckhoff_EKM1xxxEK1122.A_0002_EKM1101_0000_0017.MMS_Acceleration_Status.Number_of_samples <-> MMS Acceleration Status/Number of samples
//     PlcTask Inputs/GVL_iXlinker.EtherCAT_Master_EKxxxx.Beckhoff_EKM1xxx.Beckhoff_EKM1xxxEK1122.A_0002_EKM1101_0000_0017.MMS_Acceleration_X_Axis.Value <-> MMS Acceleration X-Axis/Value
//     PlcTask Inputs/GVL_iXlinker.EtherCAT_Master_EKxxxx.Beckhoff_EKM1xxx.Beckhoff_EKM1xxxEK1122.A_0002_EKM1101_0000_0017.MMS_Acceleration_Y_Axis.Value <-> MMS Acceleration Y-Axis/Value
//     PlcTask Inputs/GVL_iXlinker.EtherCAT_Master_EKxxxx.Beckhoff_EKM1xxx.Beckhoff_EKM1xxxEK1122.A_0002_EKM1101_0000_0017.MMS_Acceleration_Z_Axis.Value <-> MMS Acceleration Z-Axis/Value
//     PlcTask Inputs/GVL_iXlinker.EtherCAT_Master_EKxxxx.Beckhoff_EKM1xxx.Beckhoff_EKM1xxxEK1122.A_0002_EKM1101_0000_0017.MMS_Acceleration_Timestamp.Timestamp <-> MMS Acceleration Timestamp/Timestamp
//     PlcTask Inputs/GVL_iXlinker.EtherCAT_Master_EKxxxx.Beckhoff_EKM1xxx.Beckhoff_EKM1xxxEK1122.A_0002_EKM1101_0000_0017.MMS_Voltage_Us_In_Inputs.Status/Underrange <-> MMS Voltage Us In Inputs/Status/Underrange
//     PlcTask Inputs/GVL_iXlinker.EtherCAT_Master_EKxxxx.Beckhoff_EKM1xxx.Beckhoff_EKM1xxxEK1122.A_0002_EKM1101_0000_0017.MMS_Voltage_Us_In_Inputs.Status/Overrange <-> MMS Voltage Us In Inputs/Status/Overrange
//     PlcTask Inputs/GVL_iXlinker.EtherCAT_Master_EKxxxx.Beckhoff_EKM1xxx.Beckhoff_EKM1xxxEK1122.A_0002_EKM1101_0000_0017.MMS_Voltage_Us_In_Inputs.Status/Limit_1 <-> MMS Voltage Us In Inputs/Status/Limit 1
//     PlcTask Inputs/GVL_iXlinker.EtherCAT_Master_EKxxxx.Beckhoff_EKM1xxx.Beckhoff_EKM1xxxEK1122.A_0002_EKM1101_0000_0017.MMS_Voltage_Us_In_Inputs.Status/Limit_2 <-> MMS Voltage Us In Inputs/Status/Limit 2
//     PlcTask Inputs/GVL_iXlinker.EtherCAT_Master_EKxxxx.Beckhoff_EKM1xxx.Beckhoff_EKM1xxxEK1122.A_0002_EKM1101_0000_0017.MMS_Voltage_Us_In_Inputs.Status/Error <-> MMS Voltage Us In Inputs/Status/Error
//     PlcTask Inputs/GVL_iXlinker.EtherCAT_Master_EKxxxx.Beckhoff_EKM1xxx.Beckhoff_EKM1xxxEK1122.A_0002_EKM1101_0000_0017.MMS_Voltage_Us_In_Inputs.Status/TxPDO_State <-> MMS Voltage Us In Inputs/Status/TxPDO State
//     PlcTask Inputs/GVL_iXlinker.EtherCAT_Master_EKxxxx.Beckhoff_EKM1xxx.Beckhoff_EKM1xxxEK1122.A_0002_EKM1101_0000_0017.MMS_Voltage_Us_In_Inputs.Status/TxPDO_Toggle <-> MMS Voltage Us In Inputs/Status/TxPDO Toggle
//     PlcTask Inputs/GVL_iXlinker.EtherCAT_Master_EKxxxx.Beckhoff_EKM1xxx.Beckhoff_EKM1xxxEK1122.A_0002_EKM1101_0000_0017.MMS_Voltage_Us_In_Inputs.Value <-> MMS Voltage Us In Inputs/Value
//     PlcTask Inputs/GVL_iXlinker.EtherCAT_Master_EKxxxx.Beckhoff_EKM1xxx.Beckhoff_EKM1xxxEK1122.A_0002_EKM1101_0000_0017.MMS_Voltage_Up_In_Inputs.Status/Underrange <-> MMS Voltage Up In Inputs/Status/Underrange
//     PlcTask Inputs/GVL_iXlinker.EtherCAT_Master_EKxxxx.Beckhoff_EKM1xxx.Beckhoff_EKM1xxxEK1122.A_0002_EKM1101_0000_0017.MMS_Voltage_Up_In_Inputs.Status/Overrange <-> MMS Voltage Up In Inputs/Status/Overrange
//     PlcTask Inputs/GVL_iXlinker.EtherCAT_Master_EKxxxx.Beckhoff_EKM1xxx.Beckhoff_EKM1xxxEK1122.A_0002_EKM1101_0000_0017.MMS_Voltage_Up_In_Inputs.Status/Limit_1 <-> MMS Voltage Up In Inputs/Status/Limit 1
//     PlcTask Inputs/GVL_iXlinker.EtherCAT_Master_EKxxxx.Beckhoff_EKM1xxx.Beckhoff_EKM1xxxEK1122.A_0002_EKM1101_0000_0017.MMS_Voltage_Up_In_Inputs.Status/Limit_2 <-> MMS Voltage Up In Inputs/Status/Limit 2
//     PlcTask Inputs/GVL_iXlinker.EtherCAT_Master_EKxxxx.Beckhoff_EKM1xxx.Beckhoff_EKM1xxxEK1122.A_0002_EKM1101_0000_0017.MMS_Voltage_Up_In_Inputs.Status/Error <-> MMS Voltage Up In Inputs/Status/Error
//     PlcTask Inputs/GVL_iXlinker.EtherCAT_Master_EKxxxx.Beckhoff_EKM1xxx.Beckhoff_EKM1xxxEK1122.A_0002_EKM1101_0000_0017.MMS_Voltage_Up_In_Inputs.Status/TxPDO_State <-> MMS Voltage Up In Inputs/Status/TxPDO State
//     PlcTask Inputs/GVL_iXlinker.EtherCAT_Master_EKxxxx.Beckhoff_EKM1xxx.Beckhoff_EKM1xxxEK1122.A_0002_EKM1101_0000_0017.MMS_Voltage_Up_In_Inputs.Status/TxPDO_Toggle <-> MMS Voltage Up In Inputs/Status/TxPDO Toggle
//     PlcTask Inputs/GVL_iXlinker.EtherCAT_Master_EKxxxx.Beckhoff_EKM1xxx.Beckhoff_EKM1xxxEK1122.A_0002_EKM1101_0000_0017.MMS_Voltage_Up_In_Inputs.Value <-> MMS Voltage Up In Inputs/Value
//     PlcTask Inputs/GVL_iXlinker.EtherCAT_Master_EKxxxx.Beckhoff_EKM1xxx.Beckhoff_EKM1xxxEK1122.A_0002_EKM1101_0000_0017.MMS_Voltage_Up_Out_Inputs.Status/Underrange <-> MMS Voltage Up Out Inputs/Status/Underrange
//     PlcTask Inputs/GVL_iXlinker.EtherCAT_Master_EKxxxx.Beckhoff_EKM1xxx.Beckhoff_EKM1xxxEK1122.A_0002_EKM1101_0000_0017.MMS_Voltage_Up_Out_Inputs.Status/Overrange <-> MMS Voltage Up Out Inputs/Status/Overrange
//     PlcTask Inputs/GVL_iXlinker.EtherCAT_Master_EKxxxx.Beckhoff_EKM1xxx.Beckhoff_EKM1xxxEK1122.A_0002_EKM1101_0000_0017.MMS_Voltage_Up_Out_Inputs.Status/Limit_1 <-> MMS Voltage Up Out Inputs/Status/Limit 1
//     PlcTask Inputs/GVL_iXlinker.EtherCAT_Master_EKxxxx.Beckhoff_EKM1xxx.Beckhoff_EKM1xxxEK1122.A_0002_EKM1101_0000_0017.MMS_Voltage_Up_Out_Inputs.Status/Limit_2 <-> MMS Voltage Up Out Inputs/Status/Limit 2
//     PlcTask Inputs/GVL_iXlinker.EtherCAT_Master_EKxxxx.Beckhoff_EKM1xxx.Beckhoff_EKM1xxxEK1122.A_0002_EKM1101_0000_0017.MMS_Voltage_Up_Out_Inputs.Status/Error <-> MMS Voltage Up Out Inputs/Status/Error
//     PlcTask Inputs/GVL_iXlinker.EtherCAT_Master_EKxxxx.Beckhoff_EKM1xxx.Beckhoff_EKM1xxxEK1122.A_0002_EKM1101_0000_0017.MMS_Voltage_Up_Out_Inputs.Status/TxPDO_State <-> MMS Voltage Up Out Inputs/Status/TxPDO State
//     PlcTask Inputs/GVL_iXlinker.EtherCAT_Master_EKxxxx.Beckhoff_EKM1xxx.Beckhoff_EKM1xxxEK1122.A_0002_EKM1101_0000_0017.MMS_Voltage_Up_Out_Inputs.Status/TxPDO_Toggle <-> MMS Voltage Up Out Inputs/Status/TxPDO Toggle
//     PlcTask Inputs/GVL_iXlinker.EtherCAT_Master_EKxxxx.Beckhoff_EKM1xxx.Beckhoff_EKM1xxxEK1122.A_0002_EKM1101_0000_0017.MMS_Voltage_Up_Out_Inputs.Value <-> MMS Voltage Up Out Inputs/Value
//     PlcTask Outputs/GVL_iXlinker.EtherCAT_Master_EKxxxx.Beckhoff_EKM1xxx.Beckhoff_EKM1xxxEK1122.A_0002_EKM1101_0000_0017.MMS_Device_Outputs.Control/Up_Out_OFF <-> MMS Device Outputs/Control/Up Out OFF
//     PlcTask Inputs/GVL_iXlinker.EtherCAT_Master_EKxxxx.Beckhoff_EKM1xxx.Beckhoff_EKM1xxxEK1122.A_0002_EKM1101_0000_0017.WcState.WcState <-> WcState/WcState
//     PlcTask Inputs/GVL_iXlinker.EtherCAT_Master_EKxxxx.Beckhoff_EKM1xxx.Beckhoff_EKM1xxxEK1122.A_0002_EKM1101_0000_0017.WcState.InputToggle <-> WcState/InputToggle
//     PlcTask Inputs/GVL_iXlinker.EtherCAT_Master_EKxxxx.Beckhoff_EKM1xxx.Beckhoff_EKM1xxxEK1122.A_0002_EKM1101_0000_0017.InfoData.AdsAddr <-> InfoData/AdsAddr
//     PlcTask Inputs/GVL_iXlinker.EtherCAT_Master_EKxxxx.Beckhoff_EKM1xxx.Beckhoff_EKM1xxxEK1122.A_0002_EKM1101_0000_0017.InfoData.DcOutputShift <-> InfoData/DcOutputShift
//     PlcTask Inputs/GVL_iXlinker.EtherCAT_Master_EKxxxx.Beckhoff_EKM1xxx.Beckhoff_EKM1xxxEK1122.A_0002_EKM1101_0000_0017.InfoData.DcInputShift <-> InfoData/DcInputShift
//     PlcTask Inputs/GVL_iXlinker.EtherCAT_Master_EKxxxx.Beckhoff_EKM1xxx.Beckhoff_EKM1xxxEK1122.A_0002_EKM1101_0000_0017.InfoData.State <-> InfoData/State
//   PLC/PLC Instance <-> EtherCAT Master EKxxxx/Beckhoff EKM1xxx/Beckhoff EKM1xxxEK1122/A_0003(EKM1101-0000-0018)
//     PlcTask Inputs/GVL_iXlinker.EtherCAT_Master_EKxxxx.Beckhoff_EKM1xxx.Beckhoff_EKM1xxxEK1122.A_0003_EKM1101_0000_0018.MMS_Device_Inputs.Status/Diag <-> MMS Device Inputs/Status/Diag
//     PlcTask Inputs/GVL_iXlinker.EtherCAT_Master_EKxxxx.Beckhoff_EKM1xxx.Beckhoff_EKM1xxxEK1122.A_0003_EKM1101_0000_0018.MMS_Device_Inputs.Status/Error <-> MMS Device Inputs/Status/Error
//     PlcTask Inputs/GVL_iXlinker.EtherCAT_Master_EKxxxx.Beckhoff_EKM1xxx.Beckhoff_EKM1xxxEK1122.A_0003_EKM1101_0000_0018.MMS_Device_Inputs.Status/Input_cycle_Counter <-> MMS Device Inputs/Status/Input cycle Counter
//     PlcTask Inputs/GVL_iXlinker.EtherCAT_Master_EKxxxx.Beckhoff_EKM1xxx.Beckhoff_EKM1xxxEK1122.A_0003_EKM1101_0000_0018.MMS_Device_Inputs.Status/TxPDO_State <-> MMS Device Inputs/Status/TxPDO State
//     PlcTask Inputs/GVL_iXlinker.EtherCAT_Master_EKxxxx.Beckhoff_EKM1xxx.Beckhoff_EKM1xxxEK1122.A_0003_EKM1101_0000_0018.MMS_Device_Inputs.Status/ID <-> MMS Device Inputs/Status/ID
//     PlcTask Inputs/GVL_iXlinker.EtherCAT_Master_EKxxxx.Beckhoff_EKM1xxx.Beckhoff_EKM1xxxEK1122.A_0003_EKM1101_0000_0018.MMS_Acceleration_Status.Status/Error <-> MMS Acceleration Status/Status/Error
//     PlcTask Inputs/GVL_iXlinker.EtherCAT_Master_EKxxxx.Beckhoff_EKM1xxx.Beckhoff_EKM1xxxEK1122.A_0003_EKM1101_0000_0018.MMS_Acceleration_Status.Status/Underrange <-> MMS Acceleration Status/Status/Underrange
//     PlcTask Inputs/GVL_iXlinker.EtherCAT_Master_EKxxxx.Beckhoff_EKM1xxx.Beckhoff_EKM1xxxEK1122.A_0003_EKM1101_0000_0018.MMS_Acceleration_Status.Status/Overrange <-> MMS Acceleration Status/Status/Overrange
//     PlcTask Inputs/GVL_iXlinker.EtherCAT_Master_EKxxxx.Beckhoff_EKM1xxx.Beckhoff_EKM1xxxEK1122.A_0003_EKM1101_0000_0018.MMS_Acceleration_Status.Status/Diag <-> MMS Acceleration Status/Status/Diag
//     PlcTask Inputs/GVL_iXlinker.EtherCAT_Master_EKxxxx.Beckhoff_EKM1xxx.Beckhoff_EKM1xxxEK1122.A_0003_EKM1101_0000_0018.MMS_Acceleration_Status.Status/Sensor_Ovr <-> MMS Acceleration Status/Status/Sensor Ovr
//     PlcTask Inputs/GVL_iXlinker.EtherCAT_Master_EKxxxx.Beckhoff_EKM1xxx.Beckhoff_EKM1xxxEK1122.A_0003_EKM1101_0000_0018.MMS_Acceleration_Status.Status/Overrun <-> MMS Acceleration Status/Status/Overrun
//     PlcTask Inputs/GVL_iXlinker.EtherCAT_Master_EKxxxx.Beckhoff_EKM1xxx.Beckhoff_EKM1xxxEK1122.A_0003_EKM1101_0000_0018.MMS_Acceleration_Status.Status/TxPDO_State <-> MMS Acceleration Status/Status/TxPDO State
//     PlcTask Inputs/GVL_iXlinker.EtherCAT_Master_EKxxxx.Beckhoff_EKM1xxx.Beckhoff_EKM1xxxEK1122.A_0003_EKM1101_0000_0018.MMS_Acceleration_Status.Number_of_samples <-> MMS Acceleration Status/Number of samples
//     PlcTask Inputs/GVL_iXlinker.EtherCAT_Master_EKxxxx.Beckhoff_EKM1xxx.Beckhoff_EKM1xxxEK1122.A_0003_EKM1101_0000_0018.MMS_Acceleration_X_Axis.Value <-> MMS Acceleration X-Axis/Value
//     PlcTask Inputs/GVL_iXlinker.EtherCAT_Master_EKxxxx.Beckhoff_EKM1xxx.Beckhoff_EKM1xxxEK1122.A_0003_EKM1101_0000_0018.MMS_Acceleration_Y_Axis.Value <-> MMS Acceleration Y-Axis/Value
//     PlcTask Inputs/GVL_iXlinker.EtherCAT_Master_EKxxxx.Beckhoff_EKM1xxx.Beckhoff_EKM1xxxEK1122.A_0003_EKM1101_0000_0018.MMS_Acceleration_Z_Axis.Value <-> MMS Acceleration Z-Axis/Value
//     PlcTask Inputs/GVL_iXlinker.EtherCAT_Master_EKxxxx.Beckhoff_EKM1xxx.Beckhoff_EKM1xxxEK1122.A_0003_EKM1101_0000_0018.MMS_Acceleration_Timestamp.Timestamp <-> MMS Acceleration Timestamp/Timestamp
//     PlcTask Inputs/GVL_iXlinker.EtherCAT_Master_EKxxxx.Beckhoff_EKM1xxx.Beckhoff_EKM1xxxEK1122.A_0003_EKM1101_0000_0018.MMS_Voltage_Us_In_Inputs.Status/Underrange <-> MMS Voltage Us In Inputs/Status/Underrange
//     PlcTask Inputs/GVL_iXlinker.EtherCAT_Master_EKxxxx.Beckhoff_EKM1xxx.Beckhoff_EKM1xxxEK1122.A_0003_EKM1101_0000_0018.MMS_Voltage_Us_In_Inputs.Status/Overrange <-> MMS Voltage Us In Inputs/Status/Overrange
//     PlcTask Inputs/GVL_iXlinker.EtherCAT_Master_EKxxxx.Beckhoff_EKM1xxx.Beckhoff_EKM1xxxEK1122.A_0003_EKM1101_0000_0018.MMS_Voltage_Us_In_Inputs.Status/Limit_1 <-> MMS Voltage Us In Inputs/Status/Limit 1
//     PlcTask Inputs/GVL_iXlinker.EtherCAT_Master_EKxxxx.Beckhoff_EKM1xxx.Beckhoff_EKM1xxxEK1122.A_0003_EKM1101_0000_0018.MMS_Voltage_Us_In_Inputs.Status/Limit_2 <-> MMS Voltage Us In Inputs/Status/Limit 2
//     PlcTask Inputs/GVL_iXlinker.EtherCAT_Master_EKxxxx.Beckhoff_EKM1xxx.Beckhoff_EKM1xxxEK1122.A_0003_EKM1101_0000_0018.MMS_Voltage_Us_In_Inputs.Status/Error <-> MMS Voltage Us In Inputs/Status/Error
//     PlcTask Inputs/GVL_iXlinker.EtherCAT_Master_EKxxxx.Beckhoff_EKM1xxx.Beckhoff_EKM1xxxEK1122.A_0003_EKM1101_0000_0018.MMS_Voltage_Us_In_Inputs.Status/TxPDO_State <-> MMS Voltage Us In Inputs/Status/TxPDO State
//     PlcTask Inputs/GVL_iXlinker.EtherCAT_Master_EKxxxx.Beckhoff_EKM1xxx.Beckhoff_EKM1xxxEK1122.A_0003_EKM1101_0000_0018.MMS_Voltage_Us_In_Inputs.Status/TxPDO_Toggle <-> MMS Voltage Us In Inputs/Status/TxPDO Toggle
//     PlcTask Inputs/GVL_iXlinker.EtherCAT_Master_EKxxxx.Beckhoff_EKM1xxx.Beckhoff_EKM1xxxEK1122.A_0003_EKM1101_0000_0018.MMS_Voltage_Us_In_Inputs.Value <-> MMS Voltage Us In Inputs/Value
//     PlcTask Inputs/GVL_iXlinker.EtherCAT_Master_EKxxxx.Beckhoff_EKM1xxx.Beckhoff_EKM1xxxEK1122.A_0003_EKM1101_0000_0018.MMS_Voltage_Up_In_Inputs.Status/Underrange <-> MMS Voltage Up In Inputs/Status/Underrange
//     PlcTask Inputs/GVL_iXlinker.EtherCAT_Master_EKxxxx.Beckhoff_EKM1xxx.Beckhoff_EKM1xxxEK1122.A_0003_EKM1101_0000_0018.MMS_Voltage_Up_In_Inputs.Status/Overrange <-> MMS Voltage Up In Inputs/Status/Overrange
//     PlcTask Inputs/GVL_iXlinker.EtherCAT_Master_EKxxxx.Beckhoff_EKM1xxx.Beckhoff_EKM1xxxEK1122.A_0003_EKM1101_0000_0018.MMS_Voltage_Up_In_Inputs.Status/Limit_1 <-> MMS Voltage Up In Inputs/Status/Limit 1
//     PlcTask Inputs/GVL_iXlinker.EtherCAT_Master_EKxxxx.Beckhoff_EKM1xxx.Beckhoff_EKM1xxxEK1122.A_0003_EKM1101_0000_0018.MMS_Voltage_Up_In_Inputs.Status/Limit_2 <-> MMS Voltage Up In Inputs/Status/Limit 2
//     PlcTask Inputs/GVL_iXlinker.EtherCAT_Master_EKxxxx.Beckhoff_EKM1xxx.Beckhoff_EKM1xxxEK1122.A_0003_EKM1101_0000_0018.MMS_Voltage_Up_In_Inputs.Status/Error <-> MMS Voltage Up In Inputs/Status/Error
//     PlcTask Inputs/GVL_iXlinker.EtherCAT_Master_EKxxxx.Beckhoff_EKM1xxx.Beckhoff_EKM1xxxEK1122.A_0003_EKM1101_0000_0018.MMS_Voltage_Up_In_Inputs.Status/TxPDO_State <-> MMS Voltage Up In Inputs/Status/TxPDO State
//     PlcTask Inputs/GVL_iXlinker.EtherCAT_Master_EKxxxx.Beckhoff_EKM1xxx.Beckhoff_EKM1xxxEK1122.A_0003_EKM1101_0000_0018.MMS_Voltage_Up_In_Inputs.Status/TxPDO_Toggle <-> MMS Voltage Up In Inputs/Status/TxPDO Toggle
//     PlcTask Inputs/GVL_iXlinker.EtherCAT_Master_EKxxxx.Beckhoff_EKM1xxx.Beckhoff_EKM1xxxEK1122.A_0003_EKM1101_0000_0018.MMS_Voltage_Up_In_Inputs.Value <-> MMS Voltage Up In Inputs/Value
//     PlcTask Inputs/GVL_iXlinker.EtherCAT_Master_EKxxxx.Beckhoff_EKM1xxx.Beckhoff_EKM1xxxEK1122.A_0003_EKM1101_0000_0018.MMS_Voltage_Up_Out_Inputs.Status/Underrange <-> MMS Voltage Up Out Inputs/Status/Underrange
//     PlcTask Inputs/GVL_iXlinker.EtherCAT_Master_EKxxxx.Beckhoff_EKM1xxx.Beckhoff_EKM1xxxEK1122.A_0003_EKM1101_0000_0018.MMS_Voltage_Up_Out_Inputs.Status/Overrange <-> MMS Voltage Up Out Inputs/Status/Overrange
//     PlcTask Inputs/GVL_iXlinker.EtherCAT_Master_EKxxxx.Beckhoff_EKM1xxx.Beckhoff_EKM1xxxEK1122.A_0003_EKM1101_0000_0018.MMS_Voltage_Up_Out_Inputs.Status/Limit_1 <-> MMS Voltage Up Out Inputs/Status/Limit 1
//     PlcTask Inputs/GVL_iXlinker.EtherCAT_Master_EKxxxx.Beckhoff_EKM1xxx.Beckhoff_EKM1xxxEK1122.A_0003_EKM1101_0000_0018.MMS_Voltage_Up_Out_Inputs.Status/Limit_2 <-> MMS Voltage Up Out Inputs/Status/Limit 2
//     PlcTask Inputs/GVL_iXlinker.EtherCAT_Master_EKxxxx.Beckhoff_EKM1xxx.Beckhoff_EKM1xxxEK1122.A_0003_EKM1101_0000_0018.MMS_Voltage_Up_Out_Inputs.Status/Error <-> MMS Voltage Up Out Inputs/Status/Error
//     PlcTask Inputs/GVL_iXlinker.EtherCAT_Master_EKxxxx.Beckhoff_EKM1xxx.Beckhoff_EKM1xxxEK1122.A_0003_EKM1101_0000_0018.MMS_Voltage_Up_Out_Inputs.Status/TxPDO_State <-> MMS Voltage Up Out Inputs/Status/TxPDO State
//     PlcTask Inputs/GVL_iXlinker.EtherCAT_Master_EKxxxx.Beckhoff_EKM1xxx.Beckhoff_EKM1xxxEK1122.A_0003_EKM1101_0000_0018.MMS_Voltage_Up_Out_Inputs.Status/TxPDO_Toggle <-> MMS Voltage Up Out Inputs/Status/TxPDO Toggle
//     PlcTask Inputs/GVL_iXlinker.EtherCAT_Master_EKxxxx.Beckhoff_EKM1xxx.Beckhoff_EKM1xxxEK1122.A_0003_EKM1101_0000_0018.MMS_Voltage_Up_Out_Inputs.Value <-> MMS Voltage Up Out Inputs/Value
//     PlcTask Outputs/GVL_iXlinker.EtherCAT_Master_EKxxxx.Beckhoff_EKM1xxx.Beckhoff_EKM1xxxEK1122.A_0003_EKM1101_0000_0018.MMS_Device_Outputs.Control/Up_Out_OFF <-> MMS Device Outputs/Control/Up Out OFF
//     PlcTask Inputs/GVL_iXlinker.EtherCAT_Master_EKxxxx.Beckhoff_EKM1xxx.Beckhoff_EKM1xxxEK1122.A_0003_EKM1101_0000_0018.WcState.WcState <-> WcState/WcState
//     PlcTask Inputs/GVL_iXlinker.EtherCAT_Master_EKxxxx.Beckhoff_EKM1xxx.Beckhoff_EKM1xxxEK1122.A_0003_EKM1101_0000_0018.WcState.InputToggle <-> WcState/InputToggle
//     PlcTask Inputs/GVL_iXlinker.EtherCAT_Master_EKxxxx.Beckhoff_EKM1xxx.Beckhoff_EKM1xxxEK1122.A_0003_EKM1101_0000_0018.InfoData.AdsAddr <-> InfoData/AdsAddr
//     PlcTask Inputs/GVL_iXlinker.EtherCAT_Master_EKxxxx.Beckhoff_EKM1xxx.Beckhoff_EKM1xxxEK1122.A_0003_EKM1101_0000_0018.InfoData.DcOutputShift <-> InfoData/DcOutputShift
//     PlcTask Inputs/GVL_iXlinker.EtherCAT_Master_EKxxxx.Beckhoff_EKM1xxx.Beckhoff_EKM1xxxEK1122.A_0003_EKM1101_0000_0018.InfoData.DcInputShift <-> InfoData/DcInputShift
//     PlcTask Inputs/GVL_iXlinker.EtherCAT_Master_EKxxxx.Beckhoff_EKM1xxx.Beckhoff_EKM1xxxEK1122.A_0003_EKM1101_0000_0018.InfoData.State <-> InfoData/State
//   PLC/PLC Instance <-> EtherCAT Master EKxxxx/Beckhoff EKM1xxx/Beckhoff EKM1xxxEK1122/A_0004(EKM1101-0000-0019)
//     PlcTask Inputs/GVL_iXlinker.EtherCAT_Master_EKxxxx.Beckhoff_EKM1xxx.Beckhoff_EKM1xxxEK1122.A_0004_EKM1101_0000_0019.MMS_Device_Inputs.Status/Diag <-> MMS Device Inputs/Status/Diag
//     PlcTask Inputs/GVL_iXlinker.EtherCAT_Master_EKxxxx.Beckhoff_EKM1xxx.Beckhoff_EKM1xxxEK1122.A_0004_EKM1101_0000_0019.MMS_Device_Inputs.Status/Error <-> MMS Device Inputs/Status/Error
//     PlcTask Inputs/GVL_iXlinker.EtherCAT_Master_EKxxxx.Beckhoff_EKM1xxx.Beckhoff_EKM1xxxEK1122.A_0004_EKM1101_0000_0019.MMS_Device_Inputs.Status/Input_cycle_Counter <-> MMS Device Inputs/Status/Input cycle Counter
//     PlcTask Inputs/GVL_iXlinker.EtherCAT_Master_EKxxxx.Beckhoff_EKM1xxx.Beckhoff_EKM1xxxEK1122.A_0004_EKM1101_0000_0019.MMS_Device_Inputs.Status/TxPDO_State <-> MMS Device Inputs/Status/TxPDO State
//     PlcTask Inputs/GVL_iXlinker.EtherCAT_Master_EKxxxx.Beckhoff_EKM1xxx.Beckhoff_EKM1xxxEK1122.A_0004_EKM1101_0000_0019.MMS_Device_Inputs.Status/ID <-> MMS Device Inputs/Status/ID
//     PlcTask Inputs/GVL_iXlinker.EtherCAT_Master_EKxxxx.Beckhoff_EKM1xxx.Beckhoff_EKM1xxxEK1122.A_0004_EKM1101_0000_0019.MMS_Acceleration_Status.Status/Error <-> MMS Acceleration Status/Status/Error
//     PlcTask Inputs/GVL_iXlinker.EtherCAT_Master_EKxxxx.Beckhoff_EKM1xxx.Beckhoff_EKM1xxxEK1122.A_0004_EKM1101_0000_0019.MMS_Acceleration_Status.Status/Underrange <-> MMS Acceleration Status/Status/Underrange
//     PlcTask Inputs/GVL_iXlinker.EtherCAT_Master_EKxxxx.Beckhoff_EKM1xxx.Beckhoff_EKM1xxxEK1122.A_0004_EKM1101_0000_0019.MMS_Acceleration_Status.Status/Overrange <-> MMS Acceleration Status/Status/Overrange
//     PlcTask Inputs/GVL_iXlinker.EtherCAT_Master_EKxxxx.Beckhoff_EKM1xxx.Beckhoff_EKM1xxxEK1122.A_0004_EKM1101_0000_0019.MMS_Acceleration_Status.Status/Diag <-> MMS Acceleration Status/Status/Diag
//     PlcTask Inputs/GVL_iXlinker.EtherCAT_Master_EKxxxx.Beckhoff_EKM1xxx.Beckhoff_EKM1xxxEK1122.A_0004_EKM1101_0000_0019.MMS_Acceleration_Status.Status/Sensor_Ovr <-> MMS Acceleration Status/Status/Sensor Ovr
//     PlcTask Inputs/GVL_iXlinker.EtherCAT_Master_EKxxxx.Beckhoff_EKM1xxx.Beckhoff_EKM1xxxEK1122.A_0004_EKM1101_0000_0019.MMS_Acceleration_Status.Status/Overrun <-> MMS Acceleration Status/Status/Overrun
//     PlcTask Inputs/GVL_iXlinker.EtherCAT_Master_EKxxxx.Beckhoff_EKM1xxx.Beckhoff_EKM1xxxEK1122.A_0004_EKM1101_0000_0019.MMS_Acceleration_Status.Status/TxPDO_State <-> MMS Acceleration Status/Status/TxPDO State
//     PlcTask Inputs/GVL_iXlinker.EtherCAT_Master_EKxxxx.Beckhoff_EKM1xxx.Beckhoff_EKM1xxxEK1122.A_0004_EKM1101_0000_0019.MMS_Acceleration_Status.Number_of_samples <-> MMS Acceleration Status/Number of samples
//     PlcTask Inputs/GVL_iXlinker.EtherCAT_Master_EKxxxx.Beckhoff_EKM1xxx.Beckhoff_EKM1xxxEK1122.A_0004_EKM1101_0000_0019.MMS_Acceleration_X_Axis.Value <-> MMS Acceleration X-Axis/Value
//     PlcTask Inputs/GVL_iXlinker.EtherCAT_Master_EKxxxx.Beckhoff_EKM1xxx.Beckhoff_EKM1xxxEK1122.A_0004_EKM1101_0000_0019.MMS_Acceleration_Y_Axis.Value <-> MMS Acceleration Y-Axis/Value
//     PlcTask Inputs/GVL_iXlinker.EtherCAT_Master_EKxxxx.Beckhoff_EKM1xxx.Beckhoff_EKM1xxxEK1122.A_0004_EKM1101_0000_0019.MMS_Acceleration_Z_Axis.Value <-> MMS Acceleration Z-Axis/Value
//     PlcTask Inputs/GVL_iXlinker.EtherCAT_Master_EKxxxx.Beckhoff_EKM1xxx.Beckhoff_EKM1xxxEK1122.A_0004_EKM1101_0000_0019.MMS_Acceleration_Timestamp.Timestamp <-> MMS Acceleration Timestamp/Timestamp
//     PlcTask Inputs/GVL_iXlinker.EtherCAT_Master_EKxxxx.Beckhoff_EKM1xxx.Beckhoff_EKM1xxxEK1122.A_0004_EKM1101_0000_0019.MMS_Voltage_Us_In_Inputs.Status/Underrange <-> MMS Voltage Us In Inputs/Status/Underrange
//     PlcTask Inputs/GVL_iXlinker.EtherCAT_Master_EKxxxx.Beckhoff_EKM1xxx.Beckhoff_EKM1xxxEK1122.A_0004_EKM1101_0000_0019.MMS_Voltage_Us_In_Inputs.Status/Overrange <-> MMS Voltage Us In Inputs/Status/Overrange
//     PlcTask Inputs/GVL_iXlinker.EtherCAT_Master_EKxxxx.Beckhoff_EKM1xxx.Beckhoff_EKM1xxxEK1122.A_0004_EKM1101_0000_0019.MMS_Voltage_Us_In_Inputs.Status/Limit_1 <-> MMS Voltage Us In Inputs/Status/Limit 1
